LIN {X 0,Y 185.699,Z 175.337,A -85,B 0,C 180,E1 -22153.123,E2 -22153.123} C_VEL
LIN {X 0,Y 185.626,Z 175.353,A -85,B 0,C 180,E1 -22158.819,E2 -22158.819} C_VEL
LIN {X 0,Y 185.544,Z 175.363,A -85,B 0,C 180,E1 -22164.622,E2 -22164.622} C_VEL
LIN {X 0,Y 185.543,Z 175.355,A -85,B 0,C 180,E1 -22169.497,E2 -22169.497} C_VEL
LIN {X 0,Y 185.495,Z 175.376,A -85,B 0,C 180,E1 -22174.631,E2 -22174.631} C_VEL
LIN {X 0,Y 185.497,Z 175.355,A -85,B 0,C 180,E1 -22177.313,E2 -22177.313} C_VEL
LIN {X 0,Y 185.458,Z 175.377,A -85,B 0,C 180,E1 -22180.719,E2 -22180.719} C_VEL
LIN {X 0,Y 185.451,Z 175.371,A -85,B 0,C 180,E1 -22186.055,E2 -22186.055} C_VEL
LIN {X 0,Y 185.452,Z 175.385,A -85,B 0,C 180,E1 -22189.89,E2 -22189.89} C_VEL
LIN {X 0,Y 185.496,Z 175.378,A -85,B 0,C 180,E1 -22192.712,E2 -22192.712} C_VEL
LIN {X 0,Y 185.526,Z 175.377,A -85,B 0,C 180,E1 -22197.971,E2 -22197.971} C_VEL
LIN {X 0,Y 185.542,Z 175.364,A -85,B 0,C 180,E1 -22200.594,E2 -22200.594} C_VEL
LIN {X 0,Y 185.539,Z 175.366,A -85,B 0,C 180,E1 -22205.375,E2 -22205.375} C_VEL
LIN {X 0,Y 185.565,Z 175.425,A -85,B 0,C 180,E1 -22210.242,E2 -22210.242} C_VEL
LIN {X 0,Y 186.59,Z 178.23,A -85,B 0,C 180,E1 -22210.614,E2 -22210.614} C_VEL
LIN {X 0,Y 188.206,Z 180.509,A -85,B 0,C 180,E1 -22211.085,E2 -22211.085} C_VEL
LIN {X 0,Y 196.152,Z 194.206,A -85,B 0,C 180,E1 -22213.376,E2 -22213.376} C_VEL
LIN {X 0,Y 203.397,Z 208.041,A -85,B 0,C 180,E1 -22215.342,E2 -22215.342} C_VEL
LIN {X 0,Y 207.966,Z 220.286,A -85,B 0,C 180,E1 -22216.638,E2 -22216.638} C_VEL
LIN {X 0,Y 204.97,Z 276.924,A -85,B 0,C 180,E1 -22218.566,E2 -22218.566} C_VEL
LIN {X 0,Y 203.672,Z 290.054,A -85,B 0,C 180,E1 -22219.374,E2 -22219.374} C_VEL
LIN {X 0,Y 202.115,Z 302.14,A -85,B 0,C 180,E1 -22220.493,E2 -22220.493} C_VEL
LIN {X 0,Y 200.183,Z 313.622,A -85,B 0,C 180,E1 -22221.927,E2 -22221.927} C_VEL
LIN {X 0,Y 197.643,Z 325.508,A -85,B 0,C 180,E1 -22223.876,E2 -22223.876} C_VEL
LIN {X 0,Y 195.012,Z 336.195,A -85,B 0,C 180,E1 -22226.125,E2 -22226.125} C_VEL
LIN {X 0,Y 192.691,Z 344.89,A -85,B 0,C 180,E1 -22228.432,E2 -22228.432} C_VEL
LIN {X 0,Y 190.067,Z 353.762,A -85,B 0,C 180,E1 -22231.386,E2 -22231.386} C_VEL
LIN {X 0,Y 187.615,Z 361.86,A -85,B 0,C 180,E1 -22234.834,E2 -22234.834} C_VEL
LIN {X 0,Y 186.126,Z 366.937,A -85,B 0,C 180,E1 -22237.594,E2 -22237.594} C_VEL
LIN {X 0,Y 184.688,Z 371.865,A -85,B 0,C 180,E1 -22240.968,E2 -22240.968} C_VEL
LIN {X 0,Y 183.676,Z 375.61,A -85,B 0,C 180,E1 -22244.401,E2 -22244.401} C_VEL
LIN {X 0,Y 183.064,Z 378.261,A -85,B 0,C 180,E1 -22247.886,E2 -22247.886} C_VEL
LIN {X 0,Y 182.859,Z 379.431,A -85,B 0,C 180,E1 -22250.237,E2 -22250.237} C_VEL
LIN {X 0,Y 182.869,Z 380.191,A -85,B 0,C 180,E1 -22252.731,E2 -22252.731} C_VEL
LIN {X 0,Y 182.993,Z 380.465,A -85,B 0,C 180,E1 -22254.99,E2 -22254.99} C_VEL
LIN {X 0,Y 183.532,Z 380.08,A -85,B 0,C 180,E1 -22258.273,E2 -22258.273} C_VEL
LIN {X 0,Y 184.679,Z 378.477,A -85,B 0,C 180,E1 -22262.193,E2 -22262.193} C_VEL
LIN {X 0,Y 186.263,Z 375.796,A -85,B 0,C 180,E1 -22265.791,E2 -22265.791} C_VEL
LIN {X 0,Y 188.446,Z 371.875,A -85,B 0,C 180,E1 -22269.346,E2 -22269.346} C_VEL
LIN {X 0,Y 191.01,Z 366.954,A -85,B 0,C 180,E1 -22272.621,E2 -22272.621} C_VEL
LIN {X 0,Y 194.038,Z 360.951,A -85,B 0,C 180,E1 -22275.671,E2 -22275.671} C_VEL
LIN {X 0,Y 197.307,Z 354.042,A -85,B 0,C 180,E1 -22278.418,E2 -22278.418} C_VEL
LIN {X 0,Y 201.047,Z 345.323,A -85,B 0,C 180,E1 -22281.152,E2 -22281.152} C_VEL
LIN {X 0,Y 204.574,Z 336.068,A -85,B 0,C 180,E1 -22283.42,E2 -22283.42} C_VEL
LIN {X 0,Y 208.06,Z 325.682,A -85,B 0,C 180,E1 -22285.42,E2 -22285.42} C_VEL
LIN {X 0,Y 211.254,Z 314.574,A -85,B 0,C 180,E1 -22287.08,E2 -22287.08} C_VEL
LIN {X 0,Y 213.79,Z 303.24,A -85,B 0,C 180,E1 -22288.392,E2 -22288.392} C_VEL
LIN {X 0,Y 216.105,Z 289.683,A -85,B 0,C 180,E1 -22289.52,E2 -22289.52} C_VEL
LIN {X 0,Y 217.492,Z 277.689,A -85,B 0,C 180,E1 -22290.191,E2 -22290.191} C_VEL
LIN {X 0,Y 220.593,Z 229.858,A -85,B 0,C 180,E1 -22291.736,E2 -22291.736} C_VEL
LIN {X 0,Y 216.192,Z 219.873,A -85,B 0,C 180,E1 -22293.447,E2 -22293.447} C_VEL
LIN {X 0,Y 211.738,Z 211.762,A -85,B 0,C 180,E1 -22295.223,E2 -22295.223} C_VEL
LIN {X 0,Y 206.052,Z 202.859,A -85,B 0,C 180,E1 -22297.65,E2 -22297.65} C_VEL
LIN {X 0,Y 202.931,Z 198.41,A -85,B 0,C 180,E1 -22299.089,E2 -22299.089} C_VEL
LIN {X 0,Y 200.631,Z 195.194,A -85,B 0,C 180,E1 -22300.209,E2 -22300.209} C_VEL
LIN {X 0,Y 197.488,Z 190.877,A -85,B 0,C 180,E1 -22301.859,E2 -22301.859} C_VEL
LIN {X 0,Y 194.917,Z 187.57,A -85,B 0,C 180,E1 -22303.304,E2 -22303.304} C_VEL
LIN {X 0,Y 194.047,Z 186.236,A -85,B 0,C 180,E1 -22303.836,E2 -22303.836} C_VEL
LIN {X 0,Y 191.457,Z 183.668,A -85,B 0,C 180,E1 -22305.384,E2 -22305.384} C_VEL
LIN {X 0,Y 190.076,Z 181.021,A -85,B 0,C 180,E1 -22306.368,E2 -22306.368} C_VEL
LIN {X 0,Y 187.479,Z 179.133,A -85,B 0,C 180,E1 -22308.103,E2 -22308.103} C_VEL
LIN {X 0,Y 186.21,Z 176.799,A -85,B 0,C 180,E1 -22309.174,E2 -22309.174} C_VEL
LIN {X 0,Y 185.915,Z 175.32,A -85,B 0,C 180,E1 -22309.6,E2 -22309.6} C_VEL
LIN {X 0,Y 185.938,Z 175.322,A -85,B 0,C 180,E1 -22313.491,E2 -22313.491} C_VEL
LIN {X 0,Y 186.202,Z 175.284,A -85,B 0,C 180,E1 -22317.839,E2 -22317.839} C_VEL
LIN {X 0,Y 186.395,Z 175.246,A -85,B 0,C 180,E1 -22320.002,E2 -22320.002} C_VEL
LIN {X 0,Y 185.89,Z 175.314,A -85,B 0,C 180,E1 -22324.338,E2 -22324.338} C_VEL
LIN {X 0,Y 185.977,Z 175.315,A -85,B 0,C 180,E1 -22328.696,E2 -22328.696} C_VEL
LIN {X 0,Y 185.716,Z 175.345,A -85,B 0,C 180,E1 -22333.126,E2 -22333.126} C_VEL
LIN {X 0,Y 185.654,Z 175.346,A -85,B 0,C 180,E1 -22337.63,E2 -22337.63} C_VEL
LIN {X 0,Y 185.55,Z 175.357,A -85,B 0,C 180,E1 -22342.259,E2 -22342.259} C_VEL
LIN {X 0,Y 185.503,Z 175.365,A -85,B 0,C 180,E1 -22347.043,E2 -22347.043} C_VEL
LIN {X 0,Y 185.54,Z 175.424,A -85,B 0,C 180,E1 -22349.814,E2 -22349.814} C_VEL
LIN {X 0,Y 186.341,Z 177.863,A -85,B 0,C 180,E1 -22352.539,E2 -22352.539} C_VEL
LIN {X 0,Y 189.581,Z 182.629,A -85,B 0,C 180,E1 -22354.994,E2 -22354.994} C_VEL
LIN {X 0,Y 191.576,Z 185.013,A -85,B 0,C 180,E1 -22356.299,E2 -22356.299} C_VEL
LIN {X 0,Y 195.201,Z 190.145,A -85,B 0,C 180,E1 -22358.541,E2 -22358.541} C_VEL
LIN {X 0,Y 199.91,Z 197.428,A -85,B 0,C 180,E1 -22361.155,E2 -22361.155} C_VEL
LIN {X 0,Y 203.955,Z 204.171,A -85,B 0,C 180,E1 -22363.174,E2 -22363.174} C_VEL
LIN {X 0,Y 210.031,Z 215.033,A -85,B 0,C 180,E1 -22365.927,E2 -22365.927} C_VEL
LIN {X 0,Y 215.137,Z 226.03,A -85,B 0,C 180,E1 -22368.08,E2 -22368.08} C_VEL
LIN {X 0,Y 219.014,Z 236.011,A -85,B 0,C 180,E1 -22369.657,E2 -22369.657} C_VEL
LIN {X 0,Y 219.795,Z 245.363,A -85,B 0,C 180,E1 -22370.312,E2 -22370.312} C_VEL
LIN {X 0,Y 218.586,Z 264.433,A -85,B 0,C 180,E1 -22370.91,E2 -22370.91} C_VEL
LIN {X 0,Y 217.803,Z 270.281,A -85,B 0,C 180,E1 -22370.975,E2 -22370.975} C_VEL
LIN {X 0,Y 212.429,Z 289.298,A -85,B 0,C 180,E1 -22370.579,E2 -22370.579} C_VEL
LIN {X 0,Y 211.21,Z 295.05,A -85,B 0,C 180,E1 -22370.728,E2 -22370.728} C_VEL
LIN {X 0,Y 208.808,Z 308.904,A -85,B 0,C 180,E1 -22371.643,E2 -22371.643} C_VEL
LIN {X 0,Y 206.13,Z 320.49,A -85,B 0,C 180,E1 -22372.758,E2 -22372.758} C_VEL
LIN {X 0,Y 202.791,Z 331.818,A -85,B 0,C 180,E1 -22374.209,E2 -22374.209} C_VEL
LIN {X 0,Y 198.902,Z 343.336,A -85,B 0,C 180,E1 -22376.186,E2 -22376.186} C_VEL
LIN {X 0,Y 194.798,Z 353.604,A -85,B 0,C 180,E1 -22378.457,E2 -22378.457} C_VEL
LIN {X 0,Y 190.425,Z 363.452,A -85,B 0,C 180,E1 -22381.329,E2 -22381.329} C_VEL
LIN {X 0,Y 186.604,Z 371.647,A -85,B 0,C 180,E1 -22384.454,E2 -22384.454} C_VEL
LIN {X 0,Y 183.563,Z 377.81,A -85,B 0,C 180,E1 -22387.489,E2 -22387.489} C_VEL
LIN {X 0,Y 180.871,Z 382.939,A -85,B 0,C 180,E1 -22390.715,E2 -22390.715} C_VEL
LIN {X 0,Y 178.672,Z 386.953,A -85,B 0,C 180,E1 -22394.018,E2 -22394.018} C_VEL
LIN {X 0,Y 176.949,Z 390.71,A -85,B 0,C 180,E1 -22398.546,E2 -22398.546} C_VEL
LIN {X 0,Y 176.403,Z 391.989,A -85,B 0,C 180,E1 -22400.831,E2 -22400.831} C_VEL
LIN {X 0,Y 176.087,Z 392.855,A -85,B 0,C 180,E1 -22403.124,E2 -22403.124} C_VEL
LIN {X 0,Y 175.995,Z 393.414,A -85,B 0,C 180,E1 -22406.709,E2 -22406.709} C_VEL
LIN {X 0,Y 176.204,Z 393.047,A -85,B 0,C 180,E1 -22410,E2 -22410} C_VEL
LIN {X 0,Y 176.009,Z 391.778,A -85,B 0,C 180,E1 -22413.37,E2 -22413.37} C_VEL
LIN {X 0,Y 176.268,Z 388.535,A -85,B 0,C 180,E1 -22418.022,E2 -22418.022} C_VEL
LIN {X 0,Y 176.896,Z 384.919,A -85,B 0,C 180,E1 -22421.458,E2 -22421.458} C_VEL
LIN {X 0,Y 177.989,Z 380.162,A -85,B 0,C 180,E1 -22424.872,E2 -22424.872} C_VEL
LIN {X 0,Y 180.125,Z 373.006,A -85,B 0,C 180,E1 -22428.778,E2 -22428.778} C_VEL
LIN {X 0,Y 182.316,Z 365.664,A -85,B 0,C 180,E1 -22431.887,E2 -22431.887} C_VEL
LIN {X 0,Y 184.764,Z 357.175,A -85,B 0,C 180,E1 -22434.735,E2 -22434.735} C_VEL
LIN {X 0,Y 187.601,Z 347.407,A -85,B 0,C 180,E1 -22437.318,E2 -22437.318} C_VEL
LIN {X 0,Y 190.493,Z 336.558,A -85,B 0,C 180,E1 -22439.568,E2 -22439.568} C_VEL
LIN {X 0,Y 192.977,Z 325.994,A -85,B 0,C 180,E1 -22441.264,E2 -22441.264} C_VEL
LIN {X 0,Y 195.479,Z 313.312,A -85,B 0,C 180,E1 -22442.789,E2 -22442.789} C_VEL
LIN {X 0,Y 197.314,Z 300.667,A -85,B 0,C 180,E1 -22443.894,E2 -22443.894} C_VEL
LIN {X 0,Y 198.573,Z 287.659,A -85,B 0,C 180,E1 -22444.628,E2 -22444.628} C_VEL
LIN {X 0,Y 200.831,Z 240.985,A -85,B 0,C 180,E1 -22446.288,E2 -22446.288} C_VEL
LIN {X 0,Y 198.726,Z 223.599,A -85,B 0,C 180,E1 -22447.42,E2 -22447.42} C_VEL
LIN {X 0,Y 192.377,Z 207.146,A -85,B 0,C 180,E1 -22449.383,E2 -22449.383} C_VEL
LIN {X 0,Y 185.747,Z 192.753,A -85,B 0,C 180,E1 -22451.466,E2 -22451.466} C_VEL
LIN {X 0,Y 180.912,Z 183.531,A -85,B 0,C 180,E1 -22453.042,E2 -22453.042} C_VEL
LIN {X 0,Y 179.45,Z 180.415,A -85,B 0,C 180,E1 -22453.567,E2 -22453.567} C_VEL
LIN {X 0,Y 178.422,Z 176.261,A -85,B 0,C 180,E1 -22456.168,E2 -22456.168} C_VEL
LIN {X 0,Y 178.392,Z 176.267,A -85,B 0,C 180,E1 -22460.923,E2 -22460.923} C_VEL
LIN {X 0,Y 178.489,Z 176.254,A -85,B 0,C 180,E1 -22466.545,E2 -22466.545} C_VEL
LIN {X 0,Y 178.448,Z 176.257,A -85,B 0,C 180,E1 -22471.794,E2 -22471.794} C_VEL
LIN {X 0,Y 178.52,Z 176.248,A -85,B 0,C 180,E1 -22474.888,E2 -22474.888} C_VEL
LIN {X 0,Y 178.61,Z 176.236,A -85,B 0,C 180,E1 -22481.65,E2 -22481.65} C_VEL
LIN {X 0,Y 178.639,Z 176.233,A -85,B 0,C 180,E1 -22486.345,E2 -22486.345} C_VEL
LIN {X 0,Y 178.908,Z 176.173,A -85,B 0,C 180,E1 -22490.958,E2 -22490.958} C_VEL
LIN {X 0,Y 179.128,Z 176.172,A -85,B 0,C 180,E1 -22497.75,E2 -22497.75} C_VEL
LIN {X 0,Y 179.348,Z 176.135,A -85,B 0,C 180,E1 -22499.998,E2 -22499.998} C_VEL
LIN {X 0,Y 178.834,Z 176.177,A -85,B 0,C 180,E1 -22504.506,E2 -22504.506} C_VEL
LIN {X 0,Y 178.907,Z 176.199,A -85,B 0,C 180,E1 -22509.039,E2 -22509.039} C_VEL
LIN {X 0,Y 178.625,Z 176.212,A -85,B 0,C 180,E1 -22513.653,E2 -22513.653} C_VEL
LIN {X 0,Y 178.555,Z 176.234,A -85,B 0,C 180,E1 -22519.15,E2 -22519.15} C_VEL
LIN {X 0,Y 178.464,Z 176.238,A -85,B 0,C 180,E1 -22525.074,E2 -22525.074} C_VEL
LIN {X 0,Y 178.459,Z 176.248,A -85,B 0,C 180,E1 -22530.792,E2 -22530.792} C_VEL
LIN {X 0,Y 178.481,Z 176.25,A -85,B 0,C 180,E1 -22534.216,E2 -22534.216} C_VEL
LIN {X 0,Y 178.384,Z 176.242,A -85,B 0,C 180,E1 -22539.075,E2 -22539.075} C_VEL
LIN {X 0,Y 178.39,Z 176.265,A -85,B 0,C 180,E1 -22542.045,E2 -22542.045} C_VEL
LIN {X 0,Y 178.388,Z 176.257,A -85,B 0,C 180,E1 -22545.163,E2 -22545.163} C_VEL
LIN {X 0,Y 178.393,Z 176.251,A -85,B 0,C 180,E1 -22548.46,E2 -22548.46} C_VEL
LIN {X 0,Y 178.414,Z 176.253,A -85,B 0,C 180,E1 -22553.78,E2 -22553.78} C_VEL
LIN {X 0,Y 178.479,Z 176.248,A -85,B 0,C 180,E1 -22556.544,E2 -22556.544} C_VEL
LIN {X 0,Y 178.434,Z 176.249,A -85,B 0,C 180,E1 -22561.793,E2 -22561.793} C_VEL
LIN {X 0,Y 178.457,Z 176.24,A -85,B 0,C 180,E1 -22566.807,E2 -22566.807} C_VEL
LIN {X 0,Y 178.465,Z 176.276,A -85,B 0,C 180,E1 -22568.576,E2 -22568.576} C_VEL
LIN {X 0,Y 179.41,Z 179.027,A -85,B 0,C 180,E1 -22568.958,E2 -22568.958} C_VEL
LIN {X 0,Y 181.14,Z 181.31,A -85,B 0,C 180,E1 -22569.499,E2 -22569.499} C_VEL
LIN {X 0,Y 189.36,Z 195.188,A -85,B 0,C 180,E1 -22572.042,E2 -22572.042} C_VEL
LIN {X 0,Y 197.797,Z 211.139,A -85,B 0,C 180,E1 -22574.458,E2 -22574.458} C_VEL
LIN {X 0,Y 201.822,Z 222.284,A -85,B 0,C 180,E1 -22575.679,E2 -22575.679} C_VEL
LIN {X 0,Y 198.758,Z 277.285,A -85,B 0,C 180,E1 -22577.595,E2 -22577.595} C_VEL
LIN {X 0,Y 197.404,Z 290.657,A -85,B 0,C 180,E1 -22578.447,E2 -22578.447} C_VEL
LIN {X 0,Y 195.681,Z 303.225,A -85,B 0,C 180,E1 -22579.654,E2 -22579.654} C_VEL
LIN {X 0,Y 193.68,Z 314.47,A -85,B 0,C 180,E1 -22581.128,E2 -22581.128} C_VEL
LIN {X 0,Y 191.164,Z 325.697,A -85,B 0,C 180,E1 -22583.025,E2 -22583.025} C_VEL
LIN {X 0,Y 188.299,Z 336.855,A -85,B 0,C 180,E1 -22585.45,E2 -22585.45} C_VEL
LIN {X 0,Y 185.886,Z 345.472,A -85,B 0,C 180,E1 -22587.833,E2 -22587.833} C_VEL
LIN {X 0,Y 183.36,Z 353.757,A -85,B 0,C 180,E1 -22590.685,E2 -22590.685} C_VEL
LIN {X 0,Y 181.001,Z 361.169,A -85,B 0,C 180,E1 -22593.896,E2 -22593.896} C_VEL
LIN {X 0,Y 179.364,Z 366.428,A -85,B 0,C 180,E1 -22596.75,E2 -22596.75} C_VEL
LIN {X 0,Y 177.796,Z 371.59,A -85,B 0,C 180,E1 -22600.304,E2 -22600.304} C_VEL
LIN {X 0,Y 176.708,Z 375.409,A -85,B 0,C 180,E1 -22603.805,E2 -22603.805} C_VEL
LIN {X 0,Y 176.127,Z 377.76,A -85,B 0,C 180,E1 -22606.738,E2 -22606.738} C_VEL
LIN {X 0,Y 175.766,Z 379.958,A -85,B 0,C 180,E1 -22611.092,E2 -22611.092} C_VEL
LIN {X 0,Y 175.81,Z 380.579,A -85,B 0,C 180,E1 -22613.562,E2 -22613.562} C_VEL
LIN {X 0,Y 176.015,Z 380.698,A -85,B 0,C 180,E1 -22616.053,E2 -22616.053} C_VEL
LIN {X 0,Y 176.555,Z 380.315,A -85,B 0,C 180,E1 -22618.872,E2 -22618.872} C_VEL
LIN {X 0,Y 177.16,Z 379.591,A -85,B 0,C 180,E1 -22621.045,E2 -22621.045} C_VEL
LIN {X 0,Y 178.339,Z 377.895,A -85,B 0,C 180,E1 -22624.154,E2 -22624.154} C_VEL
LIN {X 0,Y 179.921,Z 375.368,A -85,B 0,C 180,E1 -22627.261,E2 -22627.261} C_VEL
LIN {X 0,Y 182.371,Z 371.207,A -85,B 0,C 180,E1 -22630.929,E2 -22630.929} C_VEL
LIN {X 0,Y 185.52,Z 365.487,A -85,B 0,C 180,E1 -22634.59,E2 -22634.59} C_VEL
LIN {X 0,Y 189.483,Z 357.992,A -85,B 0,C 180,E1 -22638.118,E2 -22638.118} C_VEL
LIN {X 0,Y 192.864,Z 350.831,A -85,B 0,C 180,E1 -22640.746,E2 -22640.746} C_VEL
LIN {X 0,Y 196.896,Z 341.505,A -85,B 0,C 180,E1 -22643.428,E2 -22643.428} C_VEL
LIN {X 0,Y 200.615,Z 331.686,A -85,B 0,C 180,E1 -22645.618,E2 -22645.618} C_VEL
LIN {X 0,Y 204.159,Z 320.87,A -85,B 0,C 180,E1 -22647.5,E2 -22647.5} C_VEL
LIN {X 0,Y 207.138,Z 309.895,A -85,B 0,C 180,E1 -22648.983,E2 -22648.983} C_VEL
LIN {X 0,Y 209.576,Z 298.487,A -85,B 0,C 180,E1 -22650.154,E2 -22650.154} C_VEL
LIN {X 0,Y 211.578,Z 285.314,A -85,B 0,C 180,E1 -22651.126,E2 -22651.126} C_VEL
LIN {X 0,Y 212.887,Z 272.862,A -85,B 0,C 180,E1 -22651.687,E2 -22651.687} C_VEL
LIN {X 0,Y 215.494,Z 232.157,A -85,B 0,C 180,E1 -22653.021,E2 -22653.021} C_VEL
LIN {X 0,Y 211.45,Z 223.085,A -85,B 0,C 180,E1 -22654.703,E2 -22654.703} C_VEL
LIN {X 0,Y 207.053,Z 215.086,A -85,B 0,C 180,E1 -22656.578,E2 -22656.578} C_VEL
LIN {X 0,Y 200.756,Z 205.257,A -85,B 0,C 180,E1 -22659.51,E2 -22659.51} C_VEL
LIN {X 0,Y 197.253,Z 200.427,A -85,B 0,C 180,E1 -22661.299,E2 -22661.299} C_VEL
LIN {X 0,Y 194.726,Z 196.808,A -85,B 0,C 180,E1 -22662.713,E2 -22662.713} C_VEL
LIN {X 0,Y 192.016,Z 193.03,A -85,B 0,C 180,E1 -22664.342,E2 -22664.342} C_VEL
LIN {X 0,Y 188.826,Z 189.361,A -85,B 0,C 180,E1 -22666.379,E2 -22666.379} C_VEL
LIN {X 0,Y 187.733,Z 187.466,A -85,B 0,C 180,E1 -22667.194,E2 -22667.194} C_VEL
LIN {X 0,Y 185.167,Z 185.137,A -85,B 0,C 180,E1 -22669.062,E2 -22669.062} C_VEL
LIN {X 0,Y 183.747,Z 182.254,A -85,B 0,C 180,E1 -22670.363,E2 -22670.363} C_VEL
LIN {X 0,Y 180.555,Z 179.962,A -85,B 0,C 180,E1 -22673.156,E2 -22673.156} C_VEL
LIN {X 0,Y 179.168,Z 177.584,A -85,B 0,C 180,E1 -22674.727,E2 -22674.727} C_VEL
LIN {X 0,Y 178.865,Z 176.185,A -85,B 0,C 180,E1 -22675.354,E2 -22675.354} C_VEL
LIN {X 0,Y 179.359,Z 176.122,A -85,B 0,C 180,E1 -22680.002,E2 -22680.002} C_VEL
LIN {X 0,Y 178.899,Z 176.18,A -85,B 0,C 180,E1 -22686.77,E2 -22686.77} C_VEL
LIN {X 0,Y 178.835,Z 176.187,A -85,B 0,C 180,E1 -22690.744,E2 -22690.744} C_VEL
LIN {X 0,Y 178.588,Z 176.221,A -85,B 0,C 180,E1 -22695.992,E2 -22695.992} C_VEL
LIN {X 0,Y 178.555,Z 176.244,A -85,B 0,C 180,E1 -22699.153,E2 -22699.153} C_VEL
LIN {X 0,Y 178.477,Z 176.247,A -85,B 0,C 180,E1 -22705.21,E2 -22705.21} C_VEL
LIN {X 0,Y 178.593,Z 176.951,A -85,B 0,C 180,E1 -22706.122,E2 -22706.122} C_VEL
LIN {X 0,Y 179.564,Z 179.274,A -85,B 0,C 180,E1 -22707.382,E2 -22707.382} C_VEL
LIN {X 0,Y 182.484,Z 182.336,A -85,B 0,C 180,E1 -22710.206,E2 -22710.206} C_VEL
LIN {X 0,Y 184.783,Z 184.988,A -85,B 0,C 180,E1 -22712.175,E2 -22712.175} C_VEL
LIN {X 0,Y 187.569,Z 189.126,A -85,B 0,C 180,E1 -22714.372,E2 -22714.372} C_VEL
LIN {X 0,Y 189.203,Z 191.197,A -85,B 0,C 180,E1 -22715.505,E2 -22715.505} C_VEL
LIN {X 0,Y 193.33,Z 197.395,A -85,B 0,C 180,E1 -22718.171,E2 -22718.171} C_VEL
LIN {X 0,Y 197.052,Z 203.358,A -85,B 0,C 180,E1 -22720.335,E2 -22720.335} C_VEL
LIN {X 0,Y 201.814,Z 211.439,A -85,B 0,C 180,E1 -22722.809,E2 -22722.809} C_VEL
LIN {X 0,Y 207.257,Z 222.099,A -85,B 0,C 180,E1 -22725.408,E2 -22725.408} C_VEL
LIN {X 0,Y 211.553,Z 231.812,A -85,B 0,C 180,E1 -22727.311,E2 -22727.311} C_VEL
LIN {X 0,Y 214.253,Z 239.251,A -85,B 0,C 180,E1 -22728.502,E2 -22728.502} C_VEL
LIN {X 0,Y 214.797,Z 245.776,A -85,B 0,C 180,E1 -22728.991,E2 -22728.991} C_VEL
LIN {X 0,Y 211.832,Z 289.491,A -85,B 0,C 180,E1 -22730.447,E2 -22730.447} C_VEL
LIN {X 0,Y 211.21,Z 295.05,A -85,B 0,C 180,E1 -22730.728,E2 -22730.728} C_VEL
LIN {X 0,Y 209.136,Z 302.593,A -85,B 0,C 180,E1 -22730.948,E2 -22730.948} C_VEL
LIN {X 0,Y 205.966,Z 309.864,A -85,B 0,C 180,E1 -22731.031,E2 -22731.031} C_VEL
LIN {X 0,Y 201.825,Z 318.808,A -85,B 0,C 180,E1 -22731.358,E2 -22731.358} C_VEL
LIN {X 0,Y 199.848,Z 324.061,A -85,B 0,C 180,E1 -22731.829,E2 -22731.829} C_VEL
LIN {X 0,Y 196.647,Z 334.056,A -85,B 0,C 180,E1 -22733.228,E2 -22733.228} C_VEL
LIN {X 0,Y 192.625,Z 345.049,A -85,B 0,C 180,E1 -22735.244,E2 -22735.244} C_VEL
LIN {X 0,Y 188.051,Z 355.788,A -85,B 0,C 180,E1 -22737.821,E2 -22737.821} C_VEL
LIN {X 0,Y 184.229,Z 363.753,A -85,B 0,C 180,E1 -22740.27,E2 -22740.27} C_VEL
LIN {X 0,Y 180.323,Z 371.593,A -85,B 0,C 180,E1 -22743.372,E2 -22743.372} C_VEL
LIN {X 0,Y 177.034,Z 377.893,A -85,B 0,C 180,E1 -22746.611,E2 -22746.611} C_VEL
LIN {X 0,Y 174.173,Z 382.943,A -85,B 0,C 180,E1 -22749.942,E2 -22749.942} C_VEL
LIN {X 0,Y 171.838,Z 386.883,A -85,B 0,C 180,E1 -22753.364,E2 -22753.364} C_VEL
LIN {X 0,Y 169.978,Z 390.573,A -85,B 0,C 180,E1 -22758.07,E2 -22758.07} C_VEL
LIN {X 0,Y 169.37,Z 391.821,A -85,B 0,C 180,E1 -22760.446,E2 -22760.446} C_VEL
LIN {X 0,Y 168.88,Z 393.056,A -85,B 0,C 180,E1 -22765.226,E2 -22765.226} C_VEL
LIN {X 0,Y 168.952,Z 393.095,A -85,B 0,C 180,E1 -22767.616,E2 -22767.616} C_VEL
LIN {X 0,Y 169.106,Z 392.746,A -85,B 0,C 180,E1 -22770,E2 -22770} C_VEL
LIN {X 0,Y 168.934,Z 391.583,A -85,B 0,C 180,E1 -22773.164,E2 -22773.164} C_VEL
LIN {X 0,Y 169.093,Z 389.081,A -85,B 0,C 180,E1 -22777.163,E2 -22777.163} C_VEL
LIN {X 0,Y 169.635,Z 385.757,A -85,B 0,C 180,E1 -22780.745,E2 -22780.745} C_VEL
LIN {X 0,Y 170.604,Z 381.325,A -85,B 0,C 180,E1 -22784.311,E2 -22784.311} C_VEL
LIN {X 0,Y 172.331,Z 375.687,A -85,B 0,C 180,E1 -22787.811,E2 -22787.811} C_VEL
LIN {X 0,Y 174.638,Z 368.618,A -85,B 0,C 180,E1 -22791.235,E2 -22791.235} C_VEL
LIN {X 0,Y 176.736,Z 361.529,A -85,B 0,C 180,E1 -22793.992,E2 -22793.992} C_VEL
LIN {X 0,Y 179.43,Z 352.575,A -85,B 0,C 180,E1 -22796.772,E2 -22796.772} C_VEL
LIN {X 0,Y 182.6,Z 341.774,A -85,B 0,C 180,E1 -22799.389,E2 -22799.389} C_VEL
LIN {X 0,Y 185.409,Z 331.006,A -85,B 0,C 180,E1 -22801.413,E2 -22801.413} C_VEL
LIN {X 0,Y 188.075,Z 318.936,A -85,B 0,C 180,E1 -22803.129,E2 -22803.129} C_VEL
LIN {X 0,Y 190.318,Z 306.404,A -85,B 0,C 180,E1 -22804.435,E2 -22804.435} C_VEL
LIN {X 0,Y 191.956,Z 293.256,A -85,B 0,C 180,E1 -22805.377,E2 -22805.377} C_VEL
LIN {X 0,Y 193.117,Z 275.346,A -85,B 0,C 180,E1 -22806.123,E2 -22806.123} C_VEL
LIN {X 0,Y 194.749,Z 241.728,A -85,B 0,C 180,E1 -22807.338,E2 -22807.338} C_VEL
LIN {X 0,Y 192.871,Z 225.898,A -85,B 0,C 180,E1 -22808.415,E2 -22808.415} C_VEL
LIN {X 0,Y 186.523,Z 209.516,A -85,B 0,C 180,E1 -22810.477,E2 -22810.477} C_VEL
LIN {X 0,Y 180.642,Z 196.638,A -85,B 0,C 180,E1 -22812.437,E2 -22812.437} C_VEL
LIN {X 0,Y 174.152,Z 184.06,A -85,B 0,C 180,E1 -22814.717,E2 -22814.717} C_VEL
LIN {X 0,Y 172.064,Z 180.025,A -85,B 0,C 180,E1 -22815.546,E2 -22815.546} C_VEL
LIN {X 0,Y 171.351,Z 177.143,A -85,B 0,C 180,E1 -22817.586,E2 -22817.586} C_VEL
LIN {X 0,Y 171.365,Z 177.143,A -85,B 0,C 180,E1 -22822.033,E2 -22822.033} C_VEL
LIN {X 0,Y 171.402,Z 177.139,A -85,B 0,C 180,E1 -22825.092,E2 -22825.092} C_VEL
LIN {X 0,Y 171.414,Z 177.134,A -85,B 0,C 180,E1 -22830.526,E2 -22830.526} C_VEL
LIN {X 0,Y 171.441,Z 177.13,A -85,B 0,C 180,E1 -22835.797,E2 -22835.797} C_VEL
LIN {X 0,Y 171.512,Z 177.122,A -85,B 0,C 180,E1 -22840.862,E2 -22840.862} C_VEL
LIN {X 0,Y 171.553,Z 177.114,A -85,B 0,C 180,E1 -22845.769,E2 -22845.769} C_VEL
LIN {X 0,Y 171.847,Z 177.054,A -85,B 0,C 180,E1 -22850.583,E2 -22850.583} C_VEL
LIN {X 0,Y 171.788,Z 177.079,A -85,B 0,C 180,E1 -22855.305,E2 -22855.305} C_VEL
LIN {X 0,Y 172.313,Z 177.011,A -85,B 0,C 180,E1 -22859.998,E2 -22859.998} C_VEL
LIN {X 0,Y 171.845,Z 177.068,A -85,B 0,C 180,E1 -22866.861,E2 -22866.861} C_VEL
LIN {X 0,Y 171.768,Z 177.086,A -85,B 0,C 180,E1 -22870.891,E2 -22870.891} C_VEL
LIN {X 0,Y 171.498,Z 177.089,A -85,B 0,C 180,E1 -22876.668,E2 -22876.668} C_VEL
LIN {X 0,Y 171.479,Z 177.117,A -85,B 0,C 180,E1 -22879.497,E2 -22879.497} C_VEL
LIN {X 0,Y 171.402,Z 177.112,A -85,B 0,C 180,E1 -22885.567,E2 -22885.567} C_VEL
LIN {X 0,Y 171.416,Z 177.124,A -85,B 0,C 180,E1 -22890.57,E2 -22890.57} C_VEL
LIN {X 0,Y 171.39,Z 177.129,A -85,B 0,C 180,E1 -22895.033,E2 -22895.033} C_VEL
LIN {X 0,Y 171.34,Z 177.116,A -85,B 0,C 180,E1 -22898.799,E2 -22898.799} C_VEL
LIN {X 0,Y 171.315,Z 177.145,A -85,B 0,C 180,E1 -22904.216,E2 -22904.216} C_VEL
LIN {X 0,Y 171.326,Z 177.135,A -85,B 0,C 180,E1 -22908.978,E2 -22908.978} C_VEL
LIN {X 0,Y 171.356,Z 177.144,A -85,B 0,C 180,E1 -22912.032,E2 -22912.032} C_VEL
LIN {X 0,Y 171.393,Z 177.122,A -85,B 0,C 180,E1 -22915.091,E2 -22915.091} C_VEL
LIN {X 0,Y 171.403,Z 177.125,A -85,B 0,C 180,E1 -22920.525,E2 -22920.525} C_VEL
LIN {X 0,Y 171.398,Z 177.122,A -85,B 0,C 180,E1 -22925.792,E2 -22925.792} C_VEL
LIN {X 0,Y 171.424,Z 177.115,A -85,B 0,C 180,E1 -22926.749,E2 -22926.749} C_VEL
LIN {X 0,Y 172.488,Z 180.058,A -85,B 0,C 180,E1 -22927.23,E2 -22927.23} C_VEL
LIN {X 0,Y 174.085,Z 182.231,A -85,B 0,C 180,E1 -22927.775,E2 -22927.775} C_VEL
LIN {X 0,Y 181.537,Z 194.391,A -85,B 0,C 180,E1 -22930.264,E2 -22930.264} C_VEL
LIN {X 0,Y 190.267,Z 210.383,A -85,B 0,C 180,E1 -22932.95,E2 -22932.95} C_VEL
LIN {X 0,Y 193.307,Z 217.005,A -85,B 0,C 180,E1 -22933.862,E2 -22933.862} C_VEL
LIN {X 0,Y 195.601,Z 223.464,A -85,B 0,C 180,E1 -22934.598,E2 -22934.598} C_VEL
LIN {X 0,Y 194.287,Z 248.894,A -85,B 0,C 180,E1 -22935.5,E2 -22935.5} C_VEL
LIN {X 0,Y 192.592,Z 277.949,A -85,B 0,C 180,E1 -22936.579,E2 -22936.579} C_VEL
LIN {X 0,Y 191.17,Z 291.281,A -85,B 0,C 180,E1 -22937.459,E2 -22937.459} C_VEL
LIN {X 0,Y 189.291,Z 304.244,A -85,B 0,C 180,E1 -22938.759,E2 -22938.759} C_VEL
LIN {X 0,Y 186.84,Z 316.946,A -85,B 0,C 180,E1 -22940.527,E2 -22940.527} C_VEL
LIN {X 0,Y 184.31,Z 327.672,A -85,B 0,C 180,E1 -22942.472,E2 -22942.472} C_VEL
LIN {X 0,Y 181.629,Z 337.493,A -85,B 0,C 180,E1 -22944.727,E2 -22944.727} C_VEL
LIN {X 0,Y 178.586,Z 347.723,A -85,B 0,C 180,E1 -22947.744,E2 -22947.744} C_VEL
LIN {X 0,Y 175.723,Z 356.532,A -85,B 0,C 180,E1 -22951.062,E2 -22951.062} C_VEL
LIN {X 0,Y 173.333,Z 363.849,A -85,B 0,C 180,E1 -22954.651,E2 -22954.651} C_VEL
LIN {X 0,Y 171.49,Z 369.544,A -85,B 0,C 180,E1 -22958.246,E2 -22958.246} C_VEL
LIN {X 0,Y 170.143,Z 373.984,A -85,B 0,C 180,E1 -22961.919,E2 -22961.919} C_VEL
LIN {X 0,Y 169.482,Z 376.328,A -85,B 0,C 180,E1 -22964.406,E2 -22964.406} C_VEL
LIN {X 0,Y 168.981,Z 378.167,A -85,B 0,C 180,E1 -22966.954,E2 -22966.954} C_VEL
LIN {X 0,Y 168.726,Z 379.532,A -85,B 0,C 180,E1 -22969.464,E2 -22969.464} C_VEL
LIN {X 0,Y 168.736,Z 380.805,A -85,B 0,C 180,E1 -22973.612,E2 -22973.612} C_VEL
LIN {X 0,Y 169.095,Z 380.923,A -85,B 0,C 180,E1 -22977.205,E2 -22977.205} C_VEL
LIN {X 0,Y 169.68,Z 380.464,A -85,B 0,C 180,E1 -22979.803,E2 -22979.803} C_VEL
LIN {X 0,Y 170.478,Z 379.503,A -85,B 0,C 180,E1 -22982.406,E2 -22982.406} C_VEL
LIN {X 0,Y 171.569,Z 378.084,A -85,B 0,C 180,E1 -22984.993,E2 -22984.993} C_VEL
LIN {X 0,Y 173.668,Z 374.961,A -85,B 0,C 180,E1 -22988.831,E2 -22988.831} C_VEL
LIN {X 0,Y 176.449,Z 370.499,A -85,B 0,C 180,E1 -22992.618,E2 -22992.618} C_VEL
LIN {X 0,Y 179.888,Z 364.605,A -85,B 0,C 180,E1 -22996.284,E2 -22996.284} C_VEL
LIN {X 0,Y 184.053,Z 357.058,A -85,B 0,C 180,E1 -22999.791,E2 -22999.791} C_VEL
LIN {X 0,Y 187.81,Z 349.392,A -85,B 0,C 180,E1 -23002.528,E2 -23002.528} C_VEL
LIN {X 0,Y 192.27,Z 339.257,A -85,B 0,C 180,E1 -23005.329,E2 -23005.329} C_VEL
LIN {X 0,Y 196.206,Z 329.061,A -85,B 0,C 180,E1 -23007.503,E2 -23007.503} C_VEL
LIN {X 0,Y 200.033,Z 317.306,A -85,B 0,C 180,E1 -23009.405,E2 -23009.405} C_VEL
LIN {X 0,Y 203.022,Z 305.707,A -85,B 0,C 180,E1 -23010.856,E2 -23010.856} C_VEL
LIN {X 0,Y 205.468,Z 293.49,A -85,B 0,C 180,E1 -23011.975,E2 -23011.975} C_VEL
LIN {X 0,Y 207.19,Z 281.184,A -85,B 0,C 180,E1 -23012.75,E2 -23012.75} C_VEL
LIN {X 0,Y 208.773,Z 261.428,A -85,B 0,C 180,E1 -23013.473,E2 -23013.473} C_VEL
LIN {X 0,Y 210.567,Z 234.613,A -85,B 0,C 180,E1 -23014.357,E2 -23014.357} C_VEL
LIN {X 0,Y 206.546,Z 225.664,A -85,B 0,C 180,E1 -23016.142,E2 -23016.142} C_VEL
LIN {X 0,Y 201.875,Z 217.571,A -85,B 0,C 180,E1 -23018.303,E2 -23018.303} C_VEL
LIN {X 0,Y 197.227,Z 210.262,A -85,B 0,C 180,E1 -23020.636,E2 -23020.636} C_VEL
LIN {X 0,Y 194.111,Z 205.794,A -85,B 0,C 180,E1 -23022.35,E2 -23022.35} C_VEL
LIN {X 0,Y 191.79,Z 202.428,A -85,B 0,C 180,E1 -23023.725,E2 -23023.725} C_VEL
LIN {X 0,Y 188.862,Z 198.425,A -85,B 0,C 180,E1 -23025.592,E2 -23025.592} C_VEL
LIN {X 0,Y 186.253,Z 195.065,A -85,B 0,C 180,E1 -23027.421,E2 -23027.421} C_VEL
LIN {X 0,Y 185.379,Z 193.768,A -85,B 0,C 180,E1 -23028.088,E2 -23028.088} C_VEL
LIN {X 0,Y 182.864,Z 191.052,A -85,B 0,C 180,E1 -23030.086,E2 -23030.086} C_VEL
LIN {X 0,Y 181.508,Z 188.599,A -85,B 0,C 180,E1 -23031.373,E2 -23031.373} C_VEL
LIN {X 0,Y 178.91,Z 186.56,A -85,B 0,C 180,E1 -23033.8,E2 -23033.8} C_VEL
LIN {X 0,Y 177.38,Z 183.784,A -85,B 0,C 180,E1 -23035.692,E2 -23035.692} C_VEL
LIN {X 0,Y 177.125,Z 183.038,A -85,B 0,C 180,E1 -23036.077,E2 -23036.077} C_VEL
LIN {X 0,Y 174.395,Z 181.218,A -85,B 0,C 180,E1 -23039.858,E2 -23039.858} C_VEL
LIN {X 0,Y 172.044,Z 178.214,A -85,B 0,C 180,E1 -23045.569,E2 -23045.569} C_VEL
LIN {X 0,Y 171.846,Z 177.06,A -85,B 0,C 180,E1 -23047.049,E2 -23047.049} C_VEL
LIN {X 0,Y 171.769,Z 177.067,A -85,B 0,C 180,E1 -23050.897,E2 -23050.897} C_VEL
LIN {X 0,Y 171.625,Z 177.195,A -85,B 0,C 180,E1 -23053.621,E2 -23053.621} C_VEL
LIN {X 0,Y 172.47,Z 179.845,A -85,B 0,C 180,E1 -23057.797,E2 -23057.797} C_VEL
LIN {X 0,Y 175.155,Z 182.528,A -85,B 0,C 180,E1 -23062.969,E2 -23062.969} C_VEL
LIN {X 0,Y 176.802,Z 183.241,A -85,B 0,C 180,E1 -23065.115,E2 -23065.115} C_VEL
LIN {X 0,Y 178.176,Z 186.195,A -85,B 0,C 180,E1 -23066.977,E2 -23066.977} C_VEL
LIN {X 0,Y 181.234,Z 189.474,A -85,B 0,C 180,E1 -23070.021,E2 -23070.021} C_VEL
LIN {X 0,Y 182.736,Z 191.304,A -85,B 0,C 180,E1 -23071.362,E2 -23071.362} C_VEL
LIN {X 0,Y 185.532,Z 195.541,A -85,B 0,C 180,E1 -23073.688,E2 -23073.688} C_VEL
LIN {X 0,Y 186.965,Z 197.542,A -85,B 0,C 180,E1 -23074.75,E2 -23074.75} C_VEL
LIN {X 0,Y 190.967,Z 203.794,A -85,B 0,C 180,E1 -23077.474,E2 -23077.474} C_VEL
LIN {X 0,Y 194.259,Z 209.248,A -85,B 0,C 180,E1 -23079.485,E2 -23079.485} C_VEL
LIN {X 0,Y 198.554,Z 216.927,A -85,B 0,C 180,E1 -23081.872,E2 -23081.872} C_VEL
LIN {X 0,Y 203.429,Z 226.706,A -85,B 0,C 180,E1 -23084.342,E2 -23084.342} C_VEL
LIN {X 0,Y 207.289,Z 235.711,A -85,B 0,C 180,E1 -23086.18,E2 -23086.18} C_VEL
LIN {X 0,Y 209.547,Z 241.986,A -85,B 0,C 180,E1 -23087.238,E2 -23087.238} C_VEL
LIN {X 0,Y 209.873,Z 247.469,A -85,B 0,C 180,E1 -23087.631,E2 -23087.631} C_VEL
LIN {X 0,Y 206.937,Z 288.865,A -85,B 0,C 180,E1 -23089.028,E2 -23089.028} C_VEL
LIN {X 0,Y 204.935,Z 302.848,A -85,B 0,C 180,E1 -23089.823,E2 -23089.823} C_VEL
LIN {X 0,Y 202.253,Z 314.964,A -85,B 0,C 180,E1 -23090.803,E2 -23090.803} C_VEL
LIN {X 0,Y 199.848,Z 324.061,A -85,B 0,C 180,E1 -23091.829,E2 -23091.829} C_VEL
LIN {X 0,Y 197.712,Z 329.281,A -85,B 0,C 180,E1 -23092.359,E2 -23092.359} C_VEL
LIN {X 0,Y 192.722,Z 337.523,A -85,B 0,C 180,E1 -23093.081,E2 -23093.081} C_VEL
LIN {X 0,Y 187.525,Z 345.3,A -85,B 0,C 180,E1 -23094.042,E2 -23094.042} C_VEL
LIN {X 0,Y 185.098,Z 349.778,A -85,B 0,C 180,E1 -23094.948,E2 -23094.948} C_VEL
LIN {X 0,Y 180.443,Z 359.529,A -85,B 0,C 180,E1 -23097.62,E2 -23097.62} C_VEL
LIN {X 0,Y 175.967,Z 368.122,A -85,B 0,C 180,E1 -23100.709,E2 -23100.709} C_VEL
LIN {X 0,Y 172.019,Z 375.465,A -85,B 0,C 180,E1 -23104.226,E2 -23104.226} C_VEL
LIN {X 0,Y 168.397,Z 381.425,A -85,B 0,C 180,E1 -23107.938,E2 -23107.938} C_VEL
LIN {X 0,Y 165.806,Z 385.65,A -85,B 0,C 180,E1 -23111.464,E2 -23111.464} C_VEL
LIN {X 0,Y 163.846,Z 388.839,A -85,B 0,C 180,E1 -23115.087,E2 -23115.087} C_VEL
LIN {X 0,Y 162.991,Z 390.45,A -85,B 0,C 180,E1 -23117.55,E2 -23117.55} C_VEL
LIN {X 0,Y 162.358,Z 391.646,A -85,B 0,C 180,E1 -23120.03,E2 -23120.03} C_VEL
LIN {X 0,Y 161.799,Z 392.809,A -85,B 0,C 180,E1 -23125.017,E2 -23125.017} C_VEL
LIN {X 0,Y 161.845,Z 392.82,A -85,B 0,C 180,E1 -23127.512,E2 -23127.512} C_VEL
LIN {X 0,Y 162.012,Z 392.436,A -85,B 0,C 180,E1 -23130.001,E2 -23130.001} C_VEL
LIN {X 0,Y 161.859,Z 391.396,A -85,B 0,C 180,E1 -23132.923,E2 -23132.923} C_VEL
LIN {X 0,Y 162.017,Z 388.664,A -85,B 0,C 180,E1 -23137.478,E2 -23137.478} C_VEL
LIN {X 0,Y 162.615,Z 385.276,A -85,B 0,C 180,E1 -23141.215,E2 -23141.215} C_VEL
LIN {X 0,Y 163.689,Z 380.78,A -85,B 0,C 180,E1 -23144.929,E2 -23144.929} C_VEL
LIN {X 0,Y 165.56,Z 375.071,A -85,B 0,C 180,E1 -23148.565,E2 -23148.565} C_VEL
LIN {X 0,Y 168.005,Z 367.88,A -85,B 0,C 180,E1 -23152.117,E2 -23152.117} C_VEL
LIN {X 0,Y 169.768,Z 362.113,A -85,B 0,C 180,E1 -23154.456,E2 -23154.456} C_VEL
LIN {X 0,Y 172.469,Z 353.582,A -85,B 0,C 180,E1 -23157.286,E2 -23157.286} C_VEL
LIN {X 0,Y 175.684,Z 343.042,A -85,B 0,C 180,E1 -23160.004,E2 -23160.004} C_VEL
LIN {X 0,Y 178.975,Z 331.189,A -85,B 0,C 180,E1 -23162.346,E2 -23162.346} C_VEL
LIN {X 0,Y 181.73,Z 319.262,A -85,B 0,C 180,E1 -23164.109,E2 -23164.109} C_VEL
LIN {X 0,Y 184.066,Z 306.912,A -85,B 0,C 180,E1 -23165.443,E2 -23165.443} C_VEL
LIN {X 0,Y 185.751,Z 294.26,A -85,B 0,C 180,E1 -23166.41,E2 -23166.41} C_VEL
LIN {X 0,Y 186.812,Z 279.809,A -85,B 0,C 180,E1 -23167.076,E2 -23167.076} C_VEL
LIN {X 0,Y 188.739,Z 242.57,A -85,B 0,C 180,E1 -23168.45,E2 -23168.45} C_VEL
LIN {X 0,Y 186.996,Z 228.014,A -85,B 0,C 180,E1 -23169.485,E2 -23169.485} C_VEL
LIN {X 0,Y 180.397,Z 210.983,A -85,B 0,C 180,E1 -23171.76,E2 -23171.76} C_VEL
LIN {X 0,Y 174.04,Z 197.266,A -85,B 0,C 180,E1 -23174.03,E2 -23174.03} C_VEL
LIN {X 0,Y 167.146,Z 184.22,A -85,B 0,C 180,E1 -23176.64,E2 -23176.64} C_VEL
LIN {X 0,Y 164.919,Z 180.186,A -85,B 0,C 180,E1 -23177.529,E2 -23177.529} C_VEL
LIN {X 0,Y 164.67,Z 179.565,A -85,B 0,C 180,E1 -23177.761,E2 -23177.761} C_VEL
LIN {X 0,Y 164.3,Z 178.022,A -85,B 0,C 180,E1 -23178.875,E2 -23178.875} C_VEL
LIN {X 0,Y 164.33,Z 178.018,A -85,B 0,C 180,E1 -23184.35,E2 -23184.35} C_VEL
LIN {X 0,Y 164.375,Z 178.013,A -85,B 0,C 180,E1 -23189.129,E2 -23189.129} C_VEL
LIN {X 0,Y 164.398,Z 178.007,A -85,B 0,C 180,E1 -23194.689,E2 -23194.689} C_VEL
LIN {X 0,Y 164.421,Z 178.002,A -85,B 0,C 180,E1 -23200.116,E2 -23200.116} C_VEL
LIN {X 0,Y 164.482,Z 177.995,A -85,B 0,C 180,E1 -23205.143,E2 -23205.143} C_VEL
LIN {X 0,Y 164.768,Z 177.938,A -85,B 0,C 180,E1 -23210.174,E2 -23210.174} C_VEL
LIN {X 0,Y 164.824,Z 177.922,A -85,B 0,C 180,E1 -23212.649,E2 -23212.649} C_VEL
LIN {X 0,Y 165.277,Z 177.887,A -85,B 0,C 180,E1 -23219.998,E2 -23219.998} C_VEL
LIN {X 0,Y 164.822,Z 177.947,A -85,B 0,C 180,E1 -23227.347,E2 -23227.347} C_VEL
LIN {X 0,Y 164.703,Z 177.966,A -85,B 0,C 180,E1 -23231.056,E2 -23231.056} C_VEL
LIN {X 0,Y 164.423,Z 177.975,A -85,B 0,C 180,E1 -23237.408,E2 -23237.408} C_VEL
LIN {X 0,Y 164.42,Z 177.999,A -85,B 0,C 180,E1 -23239.994,E2 -23239.994} C_VEL
LIN {X 0,Y 164.338,Z 177.986,A -85,B 0,C 180,E1 -23246.092,E2 -23246.092} C_VEL
LIN {X 0,Y 164.356,Z 178.006,A -85,B 0,C 180,E1 -23251.215,E2 -23251.215} C_VEL
LIN {X 0,Y 164.277,Z 177.998,A -85,B 0,C 180,E1 -23256.791,E2 -23256.791} C_VEL
LIN {X 0,Y 164.283,Z 178.003,A -85,B 0,C 180,E1 -23259.916,E2 -23259.916} C_VEL
LIN {X 0,Y 164.277,Z 178.024,A -85,B 0,C 180,E1 -23263.34,E2 -23263.34} C_VEL
LIN {X 0,Y 164.256,Z 178.005,A -85,B 0,C 180,E1 -23266.796,E2 -23266.796} C_VEL
LIN {X 0,Y 164.285,Z 178.023,A -85,B 0,C 180,E1 -23270.353,E2 -23270.353} C_VEL
LIN {X 0,Y 164.321,Z 178.004,A -85,B 0,C 180,E1 -23274.349,E2 -23274.349} C_VEL
LIN {X 0,Y 164.366,Z 178.011,A -85,B 0,C 180,E1 -23279.129,E2 -23279.129} C_VEL
LIN {X 0,Y 164.357,Z 178.008,A -85,B 0,C 180,E1 -23284.766,E2 -23284.766} C_VEL
LIN {X 0,Y 165.285,Z 180.729,A -85,B 0,C 180,E1 -23285.219,E2 -23285.219} C_VEL
LIN {X 0,Y 167.274,Z 183.386,A -85,B 0,C 180,E1 -23285.961,E2 -23285.961} C_VEL
LIN {X 0,Y 176.098,Z 197.581,A -85,B 0,C 180,E1 -23289.116,E2 -23289.116} C_VEL
LIN {X 0,Y 184.31,Z 212.694,A -85,B 0,C 180,E1 -23291.809,E2 -23291.809} C_VEL
LIN {X 0,Y 187.7,Z 219.892,A -85,B 0,C 180,E1 -23292.877,E2 -23292.877} C_VEL
LIN {X 0,Y 189.698,Z 225.655,A -85,B 0,C 180,E1 -23293.554,E2 -23293.554} C_VEL
LIN {X 0,Y 186.516,Z 278.133,A -85,B 0,C 180,E1 -23295.477,E2 -23295.477} C_VEL
LIN {X 0,Y 185.068,Z 291.3,A -85,B 0,C 180,E1 -23296.363,E2 -23296.363} C_VEL
LIN {X 0,Y 183.145,Z 304.173,A -85,B 0,C 180,E1 -23297.675,E2 -23297.675} C_VEL
LIN {X 0,Y 180.769,Z 316.136,A -85,B 0,C 180,E1 -23299.357,E2 -23299.357} C_VEL
LIN {X 0,Y 177.906,Z 327.839,A -85,B 0,C 180,E1 -23301.509,E2 -23301.509} C_VEL
LIN {X 0,Y 174.994,Z 338.094,A -85,B 0,C 180,E1 -23303.948,E2 -23303.948} C_VEL
LIN {X 0,Y 171.832,Z 348.269,A -85,B 0,C 180,E1 -23307.069,E2 -23307.069} C_VEL
LIN {X 0,Y 169.248,Z 355.843,A -85,B 0,C 180,E1 -23310,E2 -23310} C_VEL
LIN {X 0,Y 166.691,Z 363.246,A -85,B 0,C 180,E1 -23313.625,E2 -23313.625} C_VEL
LIN {X 0,Y 164.713,Z 369.105,A -85,B 0,C 180,E1 -23317.354,E2 -23317.354} C_VEL
LIN {X 0,Y 163.256,Z 373.698,A -85,B 0,C 180,E1 -23321.169,E2 -23321.169} C_VEL
LIN {X 0,Y 162.224,Z 377.154,A -85,B 0,C 180,E1 -23325.066,E2 -23325.066} C_VEL
LIN {X 0,Y 161.793,Z 378.871,A -85,B 0,C 180,E1 -23327.702,E2 -23327.702} C_VEL
LIN {X 0,Y 161.6,Z 380.117,A -85,B 0,C 180,E1 -23330.36,E2 -23330.36} C_VEL
LIN {X 0,Y 161.648,Z 381.097,A -85,B 0,C 180,E1 -23334.08,E2 -23334.08} C_VEL
LIN {X 0,Y 162.228,Z 381.105,A -85,B 0,C 180,E1 -23338.459,E2 -23338.459} C_VEL
LIN {X 0,Y 162.93,Z 380.488,A -85,B 0,C 180,E1 -23341.172,E2 -23341.172} C_VEL
LIN {X 0,Y 164.836,Z 378.279,A -85,B 0,C 180,E1 -23345.899,E2 -23345.899} C_VEL
LIN {X 0,Y 166.691,Z 375.703,A -85,B 0,C 180,E1 -23349.229,E2 -23349.229} C_VEL
LIN {X 0,Y 169.578,Z 371.478,A -85,B 0,C 180,E1 -23353.143,E2 -23353.143} C_VEL
LIN {X 0,Y 173.158,Z 365.794,A -85,B 0,C 180,E1 -23356.934,E2 -23356.934} C_VEL
LIN {X 0,Y 176.832,Z 359.614,A -85,B 0,C 180,E1 -23360.059,E2 -23360.059} C_VEL
LIN {X 0,Y 180.641,Z 352.492,A -85,B 0,C 180,E1 -23362.899,E2 -23362.899} C_VEL
LIN {X 0,Y 185.318,Z 342.893,A -85,B 0,C 180,E1 -23365.855,E2 -23365.855} C_VEL
LIN {X 0,Y 189.363,Z 333.393,A -85,B 0,C 180,E1 -23368.1,E2 -23368.1} C_VEL
LIN {X 0,Y 193.514,Z 321.932,A -85,B 0,C 180,E1 -23370.188,E2 -23370.188} C_VEL
LIN {X 0,Y 196.916,Z 310.539,A -85,B 0,C 180,E1 -23371.776,E2 -23371.776} C_VEL
LIN {X 0,Y 199.732,Z 298.296,A -85,B 0,C 180,E1 -23373.05,E2 -23373.05} C_VEL
LIN {X 0,Y 201.843,Z 285.505,A -85,B 0,C 180,E1 -23373.996,E2 -23373.996} C_VEL
LIN {X 0,Y 203.217,Z 273.185,A -85,B 0,C 180,E1 -23374.554,E2 -23374.554} C_VEL
LIN {X 0,Y 205.794,Z 237.248,A -85,B 0,C 180,E1 -23375.736,E2 -23375.736} C_VEL
LIN {X 0,Y 201.978,Z 228.841,A -85,B 0,C 180,E1 -23377.573,E2 -23377.573} C_VEL
LIN {X 0,Y 196.487,Z 219.402,A -85,B 0,C 180,E1 -23380.334,E2 -23380.334} C_VEL
LIN {X 0,Y 191.843,Z 212.23,A -85,B 0,C 180,E1 -23382.96,E2 -23382.96} C_VEL
LIN {X 0,Y 188.524,Z 207.512,A -85,B 0,C 180,E1 -23385.028,E2 -23385.028} C_VEL
LIN {X 0,Y 186.634,Z 204.74,A -85,B 0,C 180,E1 -23386.338,E2 -23386.338} C_VEL
LIN {X 0,Y 183.883,Z 200.995,A -85,B 0,C 180,E1 -23388.379,E2 -23388.379} C_VEL
LIN {X 0,Y 182.789,Z 199.75,A -85,B 0,C 180,E1 -23389.245,E2 -23389.245} C_VEL
LIN {X 0,Y 180.304,Z 196.339,A -85,B 0,C 180,E1 -23391.456,E2 -23391.456} C_VEL
LIN {X 0,Y 179.631,Z 195.2,A -85,B 0,C 180,E1 -23392.131,E2 -23392.131} C_VEL
LIN {X 0,Y 177.116,Z 192.923,A -85,B 0,C 180,E1 -23394.666,E2 -23394.666} C_VEL
LIN {X 0,Y 175.439,Z 189.821,A -85,B 0,C 180,E1 -23396.938,E2 -23396.938} C_VEL
LIN {X 0,Y 171.021,Z 185.192,A -85,B 0,C 180,E1 -23405.899,E2 -23405.899} C_VEL
LIN {X 0,Y 170.85,Z 184.221,A -85,B 0,C 180,E1 -23407.091,E2 -23407.091} C_VEL
LIN {X 0,Y 170.631,Z 184.24,A -85,B 0,C 180,E1 -23413.247,E2 -23413.247} C_VEL
LIN {X 0,Y 173.334,Z 189.076,A -85,B 0,C 180,E1 -23421.649,E2 -23421.649} C_VEL
LIN {X 0,Y 175.393,Z 190.302,A -85,B 0,C 180,E1 -23424.601,E2 -23424.601} C_VEL
LIN {X 0,Y 176.919,Z 193.264,A -85,B 0,C 180,E1 -23426.706,E2 -23426.706} C_VEL
LIN {X 0,Y 179.357,Z 195.878,A -85,B 0,C 180,E1 -23429.234,E2 -23429.234} C_VEL
LIN {X 0,Y 180.735,Z 197.65,A -85,B 0,C 180,E1 -23430.539,E2 -23430.539} C_VEL
LIN {X 0,Y 183.847,Z 202.365,A -85,B 0,C 180,E1 -23433.241,E2 -23433.241} C_VEL
LIN {X 0,Y 188.151,Z 209.352,A -85,B 0,C 180,E1 -23436.43,E2 -23436.43} C_VEL
LIN {X 0,Y 191.424,Z 214.966,A -85,B 0,C 180,E1 -23438.555,E2 -23438.555} C_VEL
LIN {X 0,Y 195.559,Z 222.778,A -85,B 0,C 180,E1 -23441.015,E2 -23441.015} C_VEL
LIN {X 0,Y 199.626,Z 231.188,A -85,B 0,C 180,E1 -23443.202,E2 -23443.202} C_VEL
LIN {X 0,Y 203.233,Z 239.923,A -85,B 0,C 180,E1 -23445.057,E2 -23445.057} C_VEL
LIN {X 0,Y 204.99,Z 245.101,A -85,B 0,C 180,E1 -23445.953,E2 -23445.953} C_VEL
LIN {X 0,Y 205.094,Z 249.221,A -85,B 0,C 180,E1 -23446.219,E2 -23446.219} C_VEL
LIN {X 0,Y 202.094,Z 289.053,A -85,B 0,C 180,E1 -23447.575,E2 -23447.575} C_VEL
LIN {X 0,Y 200.015,Z 302.86,A -85,B 0,C 180,E1 -23448.371,E2 -23448.371} C_VEL
LIN {X 0,Y 197.122,Z 315.374,A -85,B 0,C 180,E1 -23449.408,E2 -23449.408} C_VEL
LIN {X 0,Y 193.481,Z 327.725,A -85,B 0,C 180,E1 -23450.867,E2 -23450.867} C_VEL
LIN {X 0,Y 189.662,Z 338.786,A -85,B 0,C 180,E1 -23452.643,E2 -23452.643} C_VEL
LIN {X 0,Y 185.526,Z 348.817,A -85,B 0,C 180,E1 -23454.712,E2 -23454.712} C_VEL
LIN {X 0,Y 185.098,Z 349.778,A -85,B 0,C 180,E1 -23454.948,E2 -23454.948} C_VEL
LIN {X 0,Y 182.595,Z 354.168,A -85,B 0,C 180,E1 -23455.941,E2 -23455.941} C_VEL
LIN {X 0,Y 176.922,Z 360.926,A -85,B 0,C 180,E1 -23457.408,E2 -23457.408} C_VEL
LIN {X 0,Y 171.18,Z 367.053,A -85,B 0,C 180,E1 -23459.112,E2 -23459.112} C_VEL
LIN {X 0,Y 168.626,Z 370.445,A -85,B 0,C 180,E1 -23460.46,E2 -23460.46} C_VEL
LIN {X 0,Y 164.78,Z 377.075,A -85,B 0,C 180,E1 -23464.008,E2 -23464.008} C_VEL
LIN {X 0,Y 160.867,Z 382.969,A -85,B 0,C 180,E1 -23468.201,E2 -23468.201} C_VEL
LIN {X 0,Y 158.265,Z 386.767,A -85,B 0,C 180,E1 -23471.89,E2 -23471.89} C_VEL
LIN {X 0,Y 156.953,Z 388.749,A -85,B 0,C 180,E1 -23474.416,E2 -23474.416} C_VEL
LIN {X 0,Y 156.021,Z 390.325,A -85,B 0,C 180,E1 -23476.984,E2 -23476.984} C_VEL
LIN {X 0,Y 154.909,Z 392.202,A -85,B 0,C 180,E1 -23482.178,E2 -23482.178} C_VEL
LIN {X 0,Y 154.745,Z 392.544,A -85,B 0,C 180,E1 -23487.397,E2 -23487.397} C_VEL
LIN {X 0,Y 154.919,Z 392.104,A -85,B 0,C 180,E1 -23490.001,E2 -23490.001} C_VEL
LIN {X 0,Y 154.781,Z 391.222,A -85,B 0,C 180,E1 -23492.603,E2 -23492.603} C_VEL
LIN {X 0,Y 154.761,Z 389.933,A -85,B 0,C 180,E1 -23495.212,E2 -23495.212} C_VEL
LIN {X 0,Y 155.149,Z 387.177,A -85,B 0,C 180,E1 -23499.123,E2 -23499.123} C_VEL
LIN {X 0,Y 155.941,Z 383.359,A -85,B 0,C 180,E1 -23503.024,E2 -23503.024} C_VEL
LIN {X 0,Y 157.415,Z 378.395,A -85,B 0,C 180,E1 -23506.871,E2 -23506.871} C_VEL
LIN {X 0,Y 159.516,Z 372.129,A -85,B 0,C 180,E1 -23510.639,E2 -23510.639} C_VEL
LIN {X 0,Y 161.664,Z 365.923,A -85,B 0,C 180,E1 -23513.604,E2 -23513.604} C_VEL
LIN {X 0,Y 164.35,Z 357.979,A -85,B 0,C 180,E1 -23516.681,E2 -23516.681} C_VEL
LIN {X 0,Y 167.431,Z 348.579,A -85,B 0,C 180,E1 -23519.553,E2 -23519.553} C_VEL
LIN {X 0,Y 170.647,Z 338.133,A -85,B 0,C 180,E1 -23522.023,E2 -23522.023} C_VEL
LIN {X 0,Y 173.788,Z 326.549,A -85,B 0,C 180,E1 -23524.133,E2 -23524.133} C_VEL
LIN {X 0,Y 176.565,Z 314.359,A -85,B 0,C 180,E1 -23525.777,E2 -23525.777} C_VEL
LIN {X 0,Y 178.711,Z 301.575,A -85,B 0,C 180,E1 -23527.027,E2 -23527.027} C_VEL
LIN {X 0,Y 180.259,Z 288.304,A -85,B 0,C 180,E1 -23527.885,E2 -23527.885} C_VEL
LIN {X 0,Y 182.749,Z 243.517,A -85,B 0,C 180,E1 -23529.613,E2 -23529.613} C_VEL
LIN {X 0,Y 181.325,Z 230.695,A -85,B 0,C 180,E1 -23530.554,E2 -23530.554} C_VEL
LIN {X 0,Y 175.284,Z 214.753,A -85,B 0,C 180,E1 -23532.781,E2 -23532.781} C_VEL
LIN {X 0,Y 169.304,Z 201.615,A -85,B 0,C 180,E1 -23535.031,E2 -23535.031} C_VEL
LIN {X 0,Y 162.591,Z 188.766,A -85,B 0,C 180,E1 -23537.722,E2 -23537.722} C_VEL
LIN {X 0,Y 159.457,Z 183.397,A -85,B 0,C 180,E1 -23539.044,E2 -23539.044} C_VEL
LIN {X 0,Y 157.697,Z 180.678,A -85,B 0,C 180,E1 -23539.803,E2 -23539.803} C_VEL
LIN {X 0,Y 157.331,Z 179.308,A -85,B 0,C 180,E1 -23540.093,E2 -23540.093} C_VEL
LIN {X 0,Y 157.263,Z 178.899,A -85,B 0,C 180,E1 -23540.473,E2 -23540.473} C_VEL
LIN {X 0,Y 157.279,Z 178.897,A -85,B 0,C 180,E1 -23544.484,E2 -23544.484} C_VEL
LIN {X 0,Y 157.288,Z 178.894,A -85,B 0,C 180,E1 -23548.101,E2 -23548.101} C_VEL
LIN {X 0,Y 157.314,Z 178.891,A -85,B 0,C 180,E1 -23553.462,E2 -23553.462} C_VEL
LIN {X 0,Y 157.364,Z 178.881,A -85,B 0,C 180,E1 -23559.7,E2 -23559.7} C_VEL
LIN {X 0,Y 157.415,Z 178.877,A -85,B 0,C 180,E1 -23564.46,E2 -23564.46} C_VEL
LIN {X 0,Y 157.69,Z 178.823,A -85,B 0,C 180,E1 -23569.729,E2 -23569.729} C_VEL
LIN {X 0,Y 157.762,Z 178.8,A -85,B 0,C 180,E1 -23572.318,E2 -23572.318} C_VEL
LIN {X 0,Y 158.239,Z 178.763,A -85,B 0,C 180,E1 -23579.998,E2 -23579.998} C_VEL
LIN {X 0,Y 157.761,Z 178.828,A -85,B 0,C 180,E1 -23587.678,E2 -23587.678} C_VEL
LIN {X 0,Y 157.632,Z 178.846,A -85,B 0,C 180,E1 -23591.222,E2 -23591.222} C_VEL
LIN {X 0,Y 157.402,Z 178.839,A -85,B 0,C 180,E1 -23595.537,E2 -23595.537} C_VEL
LIN {X 0,Y 157.304,Z 178.889,A -85,B 0,C 180,E1 -23600.94,E2 -23600.94} C_VEL
LIN {X 0,Y 157.265,Z 178.862,A -85,B 0,C 180,E1 -23606.647,E2 -23606.647} C_VEL
LIN {X 0,Y 157.266,Z 178.895,A -85,B 0,C 180,E1 -23612.427,E2 -23612.427} C_VEL
LIN {X 0,Y 157.256,Z 178.874,A -85,B 0,C 180,E1 -23616.442,E2 -23616.442} C_VEL
LIN {X 0,Y 157.187,Z 178.906,A -85,B 0,C 180,E1 -23622.115,E2 -23622.115} C_VEL
LIN {X 0,Y 157.185,Z 178.886,A -85,B 0,C 180,E1 -23627.88,E2 -23627.88} C_VEL
LIN {X 0,Y 157.254,Z 178.888,A -85,B 0,C 180,E1 -23633.554,E2 -23633.554} C_VEL
LIN {X 0,Y 157.278,Z 178.897,A -85,B 0,C 180,E1 -23638.1,E2 -23638.1} C_VEL
LIN {X 0,Y 157.252,Z 178.889,A -85,B 0,C 180,E1 -23642.526,E2 -23642.526} C_VEL
LIN {X 0,Y 158.197,Z 181.653,A -85,B 0,C 180,E1 -23643.031,E2 -23643.031} C_VEL
LIN {X 0,Y 160.283,Z 184.233,A -85,B 0,C 180,E1 -23643.876,E2 -23643.876} C_VEL
LIN {X 0,Y 162.598,Z 187.685,A -85,B 0,C 180,E1 -23644.816,E2 -23644.816} C_VEL
LIN {X 0,Y 171.474,Z 202.219,A -85,B 0,C 180,E1 -23648.191,E2 -23648.191} C_VEL
LIN {X 0,Y 179.183,Z 216.578,A -85,B 0,C 180,E1 -23650.85,E2 -23650.85} C_VEL
LIN {X 0,Y 182.493,Z 223.8,A -85,B 0,C 180,E1 -23651.961,E2 -23651.961} C_VEL
LIN {X 0,Y 183.648,Z 227.074,A -85,B 0,C 180,E1 -23652.374,E2 -23652.374} C_VEL
LIN {X 0,Y 180.473,Z 278.555,A -85,B 0,C 180,E1 -23654.326,E2 -23654.326} C_VEL
LIN {X 0,Y 178.881,Z 292.22,A -85,B 0,C 180,E1 -23655.276,E2 -23655.276} C_VEL
LIN {X 0,Y 176.859,Z 305.024,A -85,B 0,C 180,E1 -23656.645,E2 -23656.645} C_VEL
LIN {X 0,Y 174.382,Z 316.87,A -85,B 0,C 180,E1 -23658.374,E2 -23658.374} C_VEL
LIN {X 0,Y 171.442,Z 328.353,A -85,B 0,C 180,E1 -23660.562,E2 -23660.562} C_VEL
LIN {X 0,Y 168.393,Z 338.643,A -85,B 0,C 180,E1 -23663.108,E2 -23663.108} C_VEL
LIN {X 0,Y 165.092,Z 348.774,A -85,B 0,C 180,E1 -23666.338,E2 -23666.338} C_VEL
LIN {X 0,Y 162.409,Z 356.306,A -85,B 0,C 180,E1 -23669.38,E2 -23669.38} C_VEL
LIN {X 0,Y 159.752,Z 363.658,A -85,B 0,C 180,E1 -23673.152,E2 -23673.152} C_VEL
LIN {X 0,Y 158.002,Z 368.631,A -85,B 0,C 180,E1 -23676.384,E2 -23676.384} C_VEL
LIN {X 0,Y 156.382,Z 373.4,A -85,B 0,C 180,E1 -23680.356,E2 -23680.356} C_VEL
LIN {X 0,Y 155.241,Z 377.009,A -85,B 0,C 180,E1 -23684.417,E2 -23684.417} C_VEL
LIN {X 0,Y 154.594,Z 379.541,A -85,B 0,C 180,E1 -23688.555,E2 -23688.555} C_VEL
LIN {X 0,Y 154.465,Z 380.64,A -85,B 0,C 180,E1 -23691.345,E2 -23691.345} C_VEL
LIN {X 0,Y 154.606,Z 381.381,A -85,B 0,C 180,E1 -23694.618,E2 -23694.618} C_VEL
LIN {X 0,Y 155.437,Z 381.231,A -85,B 0,C 180,E1 -23699.825,E2 -23699.825} C_VEL
LIN {X 0,Y 156.285,Z 380.511,A -85,B 0,C 180,E1 -23702.658,E2 -23702.658} C_VEL
LIN {X 0,Y 158.134,Z 378.474,A -85,B 0,C 180,E1 -23706.876,E2 -23706.876} C_VEL
LIN {X 0,Y 160.652,Z 375.266,A -85,B 0,C 180,E1 -23711.01,E2 -23711.01} C_VEL
LIN {X 0,Y 163.863,Z 370.757,A -85,B 0,C 180,E1 -23715.046,E2 -23715.046} C_VEL
LIN {X 0,Y 167.835,Z 364.813,A -85,B 0,C 180,E1 -23718.915,E2 -23718.915} C_VEL
LIN {X 0,Y 172.008,Z 358.091,A -85,B 0,C 180,E1 -23722.205,E2 -23722.205} C_VEL
LIN {X 0,Y 175.983,Z 350.918,A -85,B 0,C 180,E1 -23724.953,E2 -23724.953} C_VEL
LIN {X 0,Y 180.733,Z 341.327,A -85,B 0,C 180,E1 -23727.789,E2 -23727.789} C_VEL
LIN {X 0,Y 185.311,Z 330.75,A -85,B 0,C 180,E1 -23730.174,E2 -23730.174} C_VEL
LIN {X 0,Y 188.995,Z 320.773,A -85,B 0,C 180,E1 -23731.914,E2 -23731.914} C_VEL
LIN {X 0,Y 192.43,Z 309.255,A -85,B 0,C 180,E1 -23733.482,E2 -23733.482} C_VEL
LIN {X 0,Y 195.44,Z 296.257,A -85,B 0,C 180,E1 -23734.778,E2 -23734.778} C_VEL
LIN {X 0,Y 197.48,Z 283.669,A -85,B 0,C 180,E1 -23735.663,E2 -23735.663} C_VEL
LIN {X 0,Y 198.998,Z 268.764,A -85,B 0,C 180,E1 -23736.246,E2 -23736.246} C_VEL
LIN {X 0,Y 201.175,Z 239.857,A -85,B 0,C 180,E1 -23737.2,E2 -23737.2} C_VEL
LIN {X 0,Y 197.893,Z 232.832,A -85,B 0,C 180,E1 -23738.88,E2 -23738.88} C_VEL
LIN {X 0,Y 192.594,Z 223.522,A -85,B 0,C 180,E1 -23741.777,E2 -23741.777} C_VEL
LIN {X 0,Y 188.6,Z 217.321,A -85,B 0,C 180,E1 -23744.198,E2 -23744.198} C_VEL
LIN {X 0,Y 184.517,Z 211.123,A -85,B 0,C 180,E1 -23747.047,E2 -23747.047} C_VEL
LIN {X 0,Y 181.741,Z 207.212,A -85,B 0,C 180,E1 -23749.224,E2 -23749.224} C_VEL
LIN {X 0,Y 178.585,Z 203.038,A -85,B 0,C 180,E1 -23752.085,E2 -23752.085} C_VEL
LIN {X 0,Y 177.903,Z 201.854,A -85,B 0,C 180,E1 -23752.804,E2 -23752.804} C_VEL
LIN {X 0,Y 175.503,Z 199.418,A -85,B 0,C 180,E1 -23755.408,E2 -23755.408} C_VEL
LIN {X 0,Y 174.043,Z 196.672,A -85,B 0,C 180,E1 -23757.494,E2 -23757.494} C_VEL
LIN {X 0,Y 169.956,Z 191.953,A -85,B 0,C 180,E1 -23766.532,E2 -23766.532} C_VEL
LIN {X 0,Y 169.77,Z 191.163,A -85,B 0,C 180,E1 -23767.903,E2 -23767.903} C_VEL
LIN {X 0,Y 169.657,Z 191.293,A -85,B 0,C 180,E1 -23772.962,E2 -23772.962} C_VEL
LIN {X 0,Y 172.089,Z 195.951,A -85,B 0,C 180,E1 -23781.165,E2 -23781.165} C_VEL
LIN {X 0,Y 173.946,Z 197.103,A -85,B 0,C 180,E1 -23783.973,E2 -23783.973} C_VEL
LIN {X 0,Y 175.685,Z 200.269,A -85,B 0,C 180,E1 -23786.428,E2 -23786.428} C_VEL
LIN {X 0,Y 178.044,Z 202.902,A -85,B 0,C 180,E1 -23788.957,E2 -23788.957} C_VEL
LIN {X 0,Y 179.128,Z 204.621,A -85,B 0,C 180,E1 -23790.056,E2 -23790.056} C_VEL
LIN {X 0,Y 182.342,Z 209.691,A -85,B 0,C 180,E1 -23792.946,E2 -23792.946} C_VEL
LIN {X 0,Y 185.714,Z 215.438,A -85,B 0,C 180,E1 -23795.565,E2 -23795.565} C_VEL
LIN {X 0,Y 188.878,Z 221.156,A -85,B 0,C 180,E1 -23797.757,E2 -23797.757} C_VEL
LIN {X 0,Y 192.697,Z 228.692,A -85,B 0,C 180,E1 -23800.155,E2 -23800.155} C_VEL
LIN {X 0,Y 196.702,Z 237.435,A -85,B 0,C 180,E1 -23802.454,E2 -23802.454} C_VEL
LIN {X 0,Y 200.472,Z 247.509,A -85,B 0,C 180,E1 -23804.521,E2 -23804.521} C_VEL
LIN {X 0,Y 200.542,Z 249.972,A -85,B 0,C 180,E1 -23804.695,E2 -23804.695} C_VEL
LIN {X 0,Y 197.519,Z 288.234,A -85,B 0,C 180,E1 -23805.998,E2 -23805.998} C_VEL
LIN {X 0,Y 195.362,Z 302.285,A -85,B 0,C 180,E1 -23806.808,E2 -23806.808} C_VEL
LIN {X 0,Y 192.402,Z 314.795,A -85,B 0,C 180,E1 -23807.841,E2 -23807.841} C_VEL
LIN {X 0,Y 188.613,Z 327.209,A -85,B 0,C 180,E1 -23809.302,E2 -23809.302} C_VEL
LIN {X 0,Y 185.049,Z 337.047,A -85,B 0,C 180,E1 -23810.847,E2 -23810.847} C_VEL
LIN {X 0,Y 180.74,Z 347.362,A -85,B 0,C 180,E1 -23812.936,E2 -23812.936} C_VEL
LIN {X 0,Y 176.248,Z 356.7,A -85,B 0,C 180,E1 -23815.374,E2 -23815.374} C_VEL
LIN {X 0,Y 171.302,Z 365.753,A -85,B 0,C 180,E1 -23818.46,E2 -23818.46} C_VEL
LIN {X 0,Y 168.626,Z 370.445,A -85,B 0,C 180,E1 -23820.46,E2 -23820.46} C_VEL
LIN {X 0,Y 166.136,Z 373.695,A -85,B 0,C 180,E1 -23821.92,E2 -23821.92} C_VEL
LIN {X 0,Y 160.624,Z 378.483,A -85,B 0,C 180,E1 -23824.274,E2 -23824.274} C_VEL
LIN {X 0,Y 155.26,Z 382.557,A -85,B 0,C 180,E1 -23826.917,E2 -23826.917} C_VEL
LIN {X 0,Y 153.068,Z 384.679,A -85,B 0,C 180,E1 -23828.8,E2 -23828.8} C_VEL
LIN {X 0,Y 150.088,Z 388.67,A -85,B 0,C 180,E1 -23833.683,E2 -23833.683} C_VEL
LIN {X 0,Y 149.077,Z 390.186,A -85,B 0,C 180,E1 -23836.367,E2 -23836.367} C_VEL
LIN {X 0,Y 147.863,Z 391.987,A -85,B 0,C 180,E1 -23841.803,E2 -23841.803} C_VEL
LIN {X 0,Y 147.635,Z 392.318,A -85,B 0,C 180,E1 -23844.537,E2 -23844.537} C_VEL
LIN {X 0,Y 147.693,Z 392.167,A -85,B 0,C 180,E1 -23847.888,E2 -23847.888} C_VEL
LIN {X 0,Y 147.83,Z 391.766,A -85,B 0,C 180,E1 -23850.001,E2 -23850.001} C_VEL
LIN {X 0,Y 147.681,Z 390.852,A -85,B 0,C 180,E1 -23852.728,E2 -23852.728} C_VEL
LIN {X 0,Y 147.692,Z 389.533,A -85,B 0,C 180,E1 -23855.462,E2 -23855.462} C_VEL
LIN {X 0,Y 148.122,Z 386.709,A -85,B 0,C 180,E1 -23859.56,E2 -23859.56} C_VEL
LIN {X 0,Y 148.995,Z 382.82,A -85,B 0,C 180,E1 -23863.642,E2 -23863.642} C_VEL
LIN {X 0,Y 150.595,Z 377.78,A -85,B 0,C 180,E1 -23867.659,E2 -23867.659} C_VEL
LIN {X 0,Y 152.849,Z 371.425,A -85,B 0,C 180,E1 -23871.583,E2 -23871.583} C_VEL
LIN {X 0,Y 154.73,Z 366.285,A -85,B 0,C 180,E1 -23874.13,E2 -23874.13} C_VEL
LIN {X 0,Y 157.98,Z 357.065,A -85,B 0,C 180,E1 -23877.848,E2 -23877.848} C_VEL
LIN {X 0,Y 161.628,Z 346.402,A -85,B 0,C 180,E1 -23881.089,E2 -23881.089} C_VEL
LIN {X 0,Y 165.088,Z 335.57,A -85,B 0,C 180,E1 -23883.603,E2 -23883.603} C_VEL
LIN {X 0,Y 167.947,Z 325.006,A -85,B 0,C 180,E1 -23885.495,E2 -23885.495} C_VEL
LIN {X 0,Y 170.622,Z 313.468,A -85,B 0,C 180,E1 -23887.044,E2 -23887.044} C_VEL
LIN {X 0,Y 172.886,Z 300.115,A -85,B 0,C 180,E1 -23888.355,E2 -23888.355} C_VEL
LIN {X 0,Y 174.372,Z 286.974,A -85,B 0,C 180,E1 -23889.184,E2 -23889.184} C_VEL
LIN {X 0,Y 176.856,Z 244.431,A -85,B 0,C 180,E1 -23890.854,E2 -23890.854} C_VEL
LIN {X 0,Y 175.672,Z 233.051,A -85,B 0,C 180,E1 -23891.721,E2 -23891.721} C_VEL
LIN {X 0,Y 169.785,Z 217.561,A -85,B 0,C 180,E1 -23894.008,E2 -23894.008} C_VEL
LIN {X 0,Y 164.002,Z 204.75,A -85,B 0,C 180,E1 -23896.342,E2 -23896.342} C_VEL
LIN {X 0,Y 158.111,Z 193.293,A -85,B 0,C 180,E1 -23898.863,E2 -23898.863} C_VEL
LIN {X 0,Y 155.007,Z 187.942,A -85,B 0,C 180,E1 -23900.257,E2 -23900.257} C_VEL
LIN {X 0,Y 152.773,Z 184.455,A -85,B 0,C 180,E1 -23901.289,E2 -23901.289} C_VEL
LIN {X 0,Y 150.829,Z 182.014,A -85,B 0,C 180,E1 -23902.187,E2 -23902.187} C_VEL
LIN {X 0,Y 150.171,Z 179.783,A -85,B 0,C 180,E1 -23902.637,E2 -23902.637} C_VEL
LIN {X 0,Y 150.213,Z 179.777,A -85,B 0,C 180,E1 -23907.371,E2 -23907.371} C_VEL
LIN {X 0,Y 150.243,Z 179.77,A -85,B 0,C 180,E1 -23912.721,E2 -23912.721} C_VEL
LIN {X 0,Y 150.288,Z 179.763,A -85,B 0,C 180,E1 -23919.274,E2 -23919.274} C_VEL
LIN {X 0,Y 150.32,Z 179.76,A -85,B 0,C 180,E1 -23923.706,E2 -23923.706} C_VEL
LIN {X 0,Y 150.61,Z 179.709,A -85,B 0,C 180,E1 -23929.24,E2 -23929.24} C_VEL
LIN {X 0,Y 150.685,Z 179.679,A -85,B 0,C 180,E1 -23931.955,E2 -23931.955} C_VEL
LIN {X 0,Y 151.2,Z 179.639,A -85,B 0,C 180,E1 -23939.998,E2 -23939.998} C_VEL
LIN {X 0,Y 150.7,Z 179.709,A -85,B 0,C 180,E1 -23948.04,E2 -23948.04} C_VEL
LIN {X 0,Y 150.575,Z 179.722,A -85,B 0,C 180,E1 -23951.426,E2 -23951.426} C_VEL
LIN {X 0,Y 150.307,Z 179.722,A -85,B 0,C 180,E1 -23956.29,E2 -23956.29} C_VEL
LIN {X 0,Y 150.282,Z 179.764,A -85,B 0,C 180,E1 -23960.72,E2 -23960.72} C_VEL
LIN {X 0,Y 150.183,Z 179.741,A -85,B 0,C 180,E1 -23967.234,E2 -23967.234} C_VEL
LIN {X 0,Y 150.207,Z 179.774,A -85,B 0,C 180,E1 -23972.625,E2 -23972.625} C_VEL
LIN {X 0,Y 150.166,Z 179.749,A -85,B 0,C 180,E1 -23977.472,E2 -23977.472} C_VEL
LIN {X 0,Y 150.13,Z 179.78,A -85,B 0,C 180,E1 -23981.495,E2 -23981.495} C_VEL
LIN {X 0,Y 150.123,Z 179.772,A -85,B 0,C 180,E1 -23985.393,E2 -23985.393} C_VEL
LIN {X 0,Y 150.132,Z 179.772,A -85,B 0,C 180,E1 -23989.051,E2 -23989.051} C_VEL
LIN {X 0,Y 150.171,Z 179.777,A -85,B 0,C 180,E1 -23992.708,E2 -23992.708} C_VEL
LIN {X 0,Y 150.204,Z 179.775,A -85,B 0,C 180,E1 -23997.37,E2 -23997.37} C_VEL
LIN {X 0,Y 150.192,Z 179.786,A -85,B 0,C 180,E1 -24000.029,E2 -24000.029} C_VEL
LIN {X 0,Y 151.053,Z 182.371,A -85,B 0,C 180,E1 -24000.539,E2 -24000.539} C_VEL
LIN {X 0,Y 153.453,Z 185.369,A -85,B 0,C 180,E1 -24001.629,E2 -24001.629} C_VEL
LIN {X 0,Y 155.657,Z 188.672,A -85,B 0,C 180,E1 -24002.628,E2 -24002.628} C_VEL
LIN {X 0,Y 161.293,Z 197.453,A -85,B 0,C 180,E1 -24005.012,E2 -24005.012} C_VEL
LIN {X 0,Y 167.845,Z 208.539,A -85,B 0,C 180,E1 -24007.574,E2 -24007.574} C_VEL
LIN {X 0,Y 175.492,Z 223.292,A -85,B 0,C 180,E1 -24010.328,E2 -24010.328} C_VEL
LIN {X 0,Y 177.489,Z 228.117,A -85,B 0,C 180,E1 -24011.051,E2 -24011.051} C_VEL
LIN {X 0,Y 177.724,Z 230.223,A -85,B 0,C 180,E1 -24011.214,E2 -24011.214} C_VEL
LIN {X 0,Y 174.59,Z 278.213,A -85,B 0,C 180,E1 -24013.054,E2 -24013.054} C_VEL
LIN {X 0,Y 172.939,Z 291.865,A -85,B 0,C 180,E1 -24014.003,E2 -24014.003} C_VEL
LIN {X 0,Y 170.839,Z 304.865,A -85,B 0,C 180,E1 -24015.405,E2 -24015.405} C_VEL
LIN {X 0,Y 168.065,Z 317.596,A -85,B 0,C 180,E1 -24017.317,E2 -24017.317} C_VEL
LIN {X 0,Y 165.006,Z 328.985,A -85,B 0,C 180,E1 -24019.57,E2 -24019.57} C_VEL
LIN {X 0,Y 161.835,Z 339.102,A -85,B 0,C 180,E1 -24022.168,E2 -24022.168} C_VEL
LIN {X 0,Y 158.37,Z 349.282,A -85,B 0,C 180,E1 -24025.545,E2 -24025.545} C_VEL
LIN {X 0,Y 155.581,Z 356.773,A -85,B 0,C 180,E1 -24028.705,E2 -24028.705} C_VEL
LIN {X 0,Y 152.801,Z 364.074,A -85,B 0,C 180,E1 -24032.636,E2 -24032.636} C_VEL
LIN {X 0,Y 150.656,Z 369.876,A -85,B 0,C 180,E1 -24036.697,E2 -24036.697} C_VEL
LIN {X 0,Y 149.08,Z 374.418,A -85,B 0,C 180,E1 -24040.869,E2 -24040.869} C_VEL
LIN {X 0,Y 148.279,Z 376.832,A -85,B 0,C 180,E1 -24043.708,E2 -24043.708} C_VEL
LIN {X 0,Y 147.595,Z 379.374,A -85,B 0,C 180,E1 -24047.77,E2 -24047.77} C_VEL
LIN {X 0,Y 147.378,Z 381.162,A -85,B 0,C 180,E1 -24052.426,E2 -24052.426} C_VEL
LIN {X 0,Y 147.564,Z 381.673,A -85,B 0,C 180,E1 -24055.381,E2 -24055.381} C_VEL
LIN {X 0,Y 147.985,Z 381.735,A -85,B 0,C 180,E1 -24058.353,E2 -24058.353} C_VEL
LIN {X 0,Y 148.864,Z 381.232,A -85,B 0,C 180,E1 -24061.815,E2 -24061.815} C_VEL
LIN {X 0,Y 151.094,Z 379.091,A -85,B 0,C 180,E1 -24067.206,E2 -24067.206} C_VEL
LIN {X 0,Y 153.718,Z 376.073,A -85,B 0,C 180,E1 -24071.524,E2 -24071.524} C_VEL
LIN {X 0,Y 157.083,Z 371.788,A -85,B 0,C 180,E1 -24075.713,E2 -24075.713} C_VEL
LIN {X 0,Y 161.322,Z 365.863,A -85,B 0,C 180,E1 -24079.83,E2 -24079.83} C_VEL
LIN {X 0,Y 166.068,Z 358.669,A -85,B 0,C 180,E1 -24083.521,E2 -24083.521} C_VEL
LIN {X 0,Y 170.605,Z 350.988,A -85,B 0,C 180,E1 -24086.531,E2 -24086.531} C_VEL
LIN {X 0,Y 175.579,Z 341.445,A -85,B 0,C 180,E1 -24089.383,E2 -24089.383} C_VEL
LIN {X 0,Y 180.355,Z 330.929,A -85,B 0,C 180,E1 -24091.776,E2 -24091.776} C_VEL
LIN {X 0,Y 184.378,Z 320.453,A -85,B 0,C 180,E1 -24093.605,E2 -24093.605} C_VEL
LIN {X 0,Y 188.026,Z 308.433,A -85,B 0,C 180,E1 -24095.223,E2 -24095.223} C_VEL
LIN {X 0,Y 191.133,Z 295.383,A -85,B 0,C 180,E1 -24096.487,E2 -24096.487} C_VEL
LIN {X 0,Y 193.182,Z 282.752,A -85,B 0,C 180,E1 -24097.331,E2 -24097.331} C_VEL
LIN {X 0,Y 194.926,Z 264.65,A -85,B 0,C 180,E1 -24098.01,E2 -24098.01} C_VEL
LIN {X 0,Y 196.579,Z 242.39,A -85,B 0,C 180,E1 -24098.786,E2 -24098.786} C_VEL
LIN {X 0,Y 193.067,Z 235.136,A -85,B 0,C 180,E1 -24100.74,E2 -24100.74} C_VEL
LIN {X 0,Y 188.093,Z 226.509,A -85,B 0,C 180,E1 -24103.739,E2 -24103.739} C_VEL
LIN {X 0,Y 183.924,Z 219.896,A -85,B 0,C 180,E1 -24106.624,E2 -24106.624} C_VEL
LIN {X 0,Y 181.609,Z 216.515,A -85,B 0,C 180,E1 -24108.399,E2 -24108.399} C_VEL
LIN {X 0,Y 179.008,Z 212.682,A -85,B 0,C 180,E1 -24110.659,E2 -24110.659} C_VEL
LIN {X 0,Y 176.519,Z 208.997,A -85,B 0,C 180,E1 -24113.142,E2 -24113.142} C_VEL
LIN {X 0,Y 173.392,Z 205.072,A -85,B 0,C 180,E1 -24116.902,E2 -24116.902} C_VEL
LIN {X 0,Y 172.532,Z 203.411,A -85,B 0,C 180,E1 -24118.251,E2 -24118.251} C_VEL
LIN {X 0,Y 168.91,Z 198.732,A -85,B 0,C 180,E1 -24127.173,E2 -24127.173} C_VEL
LIN {X 0,Y 168.837,Z 198.2,A -85,B 0,C 180,E1 -24127.947,E2 -24127.947} C_VEL
LIN {X 0,Y 168.707,Z 198.345,A -85,B 0,C 180,E1 -24132.783,E2 -24132.783} C_VEL
LIN {X 0,Y 170.925,Z 202.865,A -85,B 0,C 180,E1 -24140.793,E2 -24140.793} C_VEL
LIN {X 0,Y 172.533,Z 203.928,A -85,B 0,C 180,E1 -24143.354,E2 -24143.354} C_VEL
LIN {X 0,Y 174.443,Z 207.258,A -85,B 0,C 180,E1 -24146.13,E2 -24146.13} C_VEL
LIN {X 0,Y 176.685,Z 209.871,A -85,B 0,C 180,E1 -24148.623,E2 -24148.623} C_VEL
LIN {X 0,Y 179.6,Z 214.805,A -85,B 0,C 180,E1 -24151.536,E2 -24151.536} C_VEL
LIN {X 0,Y 183.484,Z 221.775,A -85,B 0,C 180,E1 -24154.792,E2 -24154.792} C_VEL
LIN {X 0,Y 186.414,Z 227.392,A -85,B 0,C 180,E1 -24156.964,E2 -24156.964} C_VEL
LIN {X 0,Y 190.682,Z 236.327,A -85,B 0,C 180,E1 -24159.775,E2 -24159.775} C_VEL
LIN {X 0,Y 194.398,Z 245.472,A -85,B 0,C 180,E1 -24162.047,E2 -24162.047} C_VEL
LIN {X 0,Y 196.08,Z 250.178,A -85,B 0,C 180,E1 -24163.027,E2 -24163.027} C_VEL
LIN {X 0,Y 193.225,Z 286.902,A -85,B 0,C 180,E1 -24164.32,E2 -24164.32} C_VEL
LIN {X 0,Y 191.164,Z 300.439,A -85,B 0,C 180,E1 -24165.073,E2 -24165.073} C_VEL
LIN {X 0,Y 188.13,Z 313.324,A -85,B 0,C 180,E1 -24166.097,E2 -24166.097} C_VEL
LIN {X 0,Y 184.474,Z 325.241,A -85,B 0,C 180,E1 -24167.45,E2 -24167.45} C_VEL
LIN {X 0,Y 180.694,Z 335.372,A -85,B 0,C 180,E1 -24168.979,E2 -24168.979} C_VEL
LIN {X 0,Y 175.643,Z 346.966,A -85,B 0,C 180,E1 -24171.303,E2 -24171.303} C_VEL
LIN {X 0,Y 171.347,Z 355.447,A -85,B 0,C 180,E1 -24173.507,E2 -24173.507} C_VEL
LIN {X 0,Y 166.951,Z 363.312,A -85,B 0,C 180,E1 -24176.098,E2 -24176.098} C_VEL
LIN {X 0,Y 162.24,Z 371.052,A -85,B 0,C 180,E1 -24179.404,E2 -24179.404} C_VEL
LIN {X 0,Y 157.702,Z 378.199,A -85,B 0,C 180,E1 -24183.535,E2 -24183.535} C_VEL
LIN {X 0,Y 154.275,Z 383.008,A -85,B 0,C 180,E1 -24187.219,E2 -24187.219} C_VEL
LIN {X 0,Y 153.068,Z 384.679,A -85,B 0,C 180,E1 -24188.8,E2 -24188.8} C_VEL
LIN {X 0,Y 151.014,Z 386.574,A -85,B 0,C 180,E1 -24190.77,E2 -24190.77} C_VEL
LIN {X 0,Y 146.38,Z 389.053,A -85,B 0,C 180,E1 -24194.015,E2 -24194.015} C_VEL
LIN {X 0,Y 142.927,Z 390.482,A -85,B 0,C 180,E1 -24196.791,E2 -24196.791} C_VEL
LIN {X 0,Y 141.299,Z 391.261,A -85,B 0,C 180,E1 -24199.062,E2 -24199.062} C_VEL
LIN {X 0,Y 141.057,Z 391.414,A -85,B 0,C 180,E1 -24199.851,E2 -24199.851} C_VEL
LIN {X 0,Y 140.554,Z 392.074,A -85,B 0,C 180,E1 -24204.261,E2 -24204.261} C_VEL
LIN {X 0,Y 140.618,Z 391.761,A -85,B 0,C 180,E1 -24208.428,E2 -24208.428} C_VEL
LIN {X 0,Y 140.631,Z 390.91,A -85,B 0,C 180,E1 -24211.755,E2 -24211.755} C_VEL
LIN {X 0,Y 140.623,Z 389.129,A -85,B 0,C 180,E1 -24215.737,E2 -24215.737} C_VEL
LIN {X 0,Y 141.086,Z 386.236,A -85,B 0,C 180,E1 -24220.041,E2 -24220.041} C_VEL
LIN {X 0,Y 142.075,Z 382.276,A -85,B 0,C 180,E1 -24224.32,E2 -24224.32} C_VEL
LIN {X 0,Y 144.191,Z 376.162,A -85,B 0,C 180,E1 -24229.209,E2 -24229.209} C_VEL
LIN {X 0,Y 146.766,Z 369.444,A -85,B 0,C 180,E1 -24233.27,E2 -24233.27} C_VEL
LIN {X 0,Y 149.204,Z 362.752,A -85,B 0,C 180,E1 -24236.492,E2 -24236.492} C_VEL
LIN {X 0,Y 152.348,Z 354.293,A -85,B 0,C 180,E1 -24239.731,E2 -24239.731} C_VEL
LIN {X 0,Y 155.9,Z 344.185,A -85,B 0,C 180,E1 -24242.75,E2 -24242.75} C_VEL
LIN {X 0,Y 159.584,Z 332.761,A -85,B 0,C 180,E1 -24245.312,E2 -24245.312} C_VEL
LIN {X 0,Y 162.595,Z 321.548,A -85,B 0,C 180,E1 -24247.239,E2 -24247.239} C_VEL
LIN {X 0,Y 165.425,Z 309.068,A -85,B 0,C 180,E1 -24248.804,E2 -24248.804} C_VEL
LIN {X 0,Y 167.503,Z 296.08,A -85,B 0,C 180,E1 -24249.945,E2 -24249.945} C_VEL
LIN {X 0,Y 168.827,Z 282.333,A -85,B 0,C 180,E1 -24250.713,E2 -24250.713} C_VEL
LIN {X 0,Y 171.045,Z 245.017,A -85,B 0,C 180,E1 -24252.192,E2 -24252.192} C_VEL
LIN {X 0,Y 169.933,Z 235.225,A -85,B 0,C 180,E1 -24252.996,E2 -24252.996} C_VEL
LIN {X 0,Y 164.475,Z 220.558,A -85,B 0,C 180,E1 -24255.274,E2 -24255.274} C_VEL
LIN {X 0,Y 158.891,Z 208.07,A -85,B 0,C 180,E1 -24257.687,E2 -24257.687} C_VEL
LIN {X 0,Y 153.109,Z 196.792,A -85,B 0,C 180,E1 -24260.33,E2 -24260.33} C_VEL
LIN {X 0,Y 150.946,Z 192.984,A -85,B 0,C 180,E1 -24261.375,E2 -24261.375} C_VEL
LIN {X 0,Y 148.477,Z 189.35,A -85,B 0,C 180,E1 -24262.573,E2 -24262.573} C_VEL
LIN {X 0,Y 146.356,Z 185.998,A -85,B 0,C 180,E1 -24263.654,E2 -24263.654} C_VEL
LIN {X 0,Y 143.946,Z 183.253,A -85,B 0,C 180,E1 -24264.867,E2 -24264.867} C_VEL
LIN {X 0,Y 143.132,Z 180.66,A -85,B 0,C 180,E1 -24265.464,E2 -24265.464} C_VEL
LIN {X 0,Y 143.115,Z 180.659,A -85,B 0,C 180,E1 -24270.586,E2 -24270.586} C_VEL
LIN {X 0,Y 143.153,Z 180.654,A -85,B 0,C 180,E1 -24273.776,E2 -24273.776} C_VEL
LIN {X 0,Y 143.251,Z 180.639,A -85,B 0,C 180,E1 -24279.912,E2 -24279.912} C_VEL
LIN {X 0,Y 143.314,Z 180.632,A -85,B 0,C 180,E1 -24285.804,E2 -24285.804} C_VEL
LIN {X 0,Y 143.536,Z 180.595,A -85,B 0,C 180,E1 -24288.703,E2 -24288.703} C_VEL
LIN {X 0,Y 143.61,Z 180.56,A -85,B 0,C 180,E1 -24291.555,E2 -24291.555} C_VEL
LIN {X 0,Y 144.158,Z 180.516,A -85,B 0,C 180,E1 -24299.998,E2 -24299.998} C_VEL
LIN {X 0,Y 143.622,Z 180.593,A -85,B 0,C 180,E1 -24308.439,E2 -24308.439} C_VEL
LIN {X 0,Y 143.499,Z 180.601,A -85,B 0,C 180,E1 -24311.612,E2 -24311.612} C_VEL
LIN {X 0,Y 143.249,Z 180.604,A -85,B 0,C 180,E1 -24317.117,E2 -24317.117} C_VEL
LIN {X 0,Y 143.219,Z 180.644,A -85,B 0,C 180,E1 -24321.191,E2 -24321.191} C_VEL
LIN {X 0,Y 143.14,Z 180.617,A -85,B 0,C 180,E1 -24327.897,E2 -24327.897} C_VEL
LIN {X 0,Y 143.136,Z 180.655,A -85,B 0,C 180,E1 -24333.414,E2 -24333.414} C_VEL
LIN {X 0,Y 143.049,Z 180.641,A -85,B 0,C 180,E1 -24339.691,E2 -24339.691} C_VEL
LIN {X 0,Y 143.048,Z 180.668,A -85,B 0,C 180,E1 -24343.454,E2 -24343.454} C_VEL
LIN {X 0,Y 143.033,Z 180.646,A -85,B 0,C 180,E1 -24347.475,E2 -24347.475} C_VEL
LIN {X 0,Y 143.068,Z 180.668,A -85,B 0,C 180,E1 -24351.807,E2 -24351.807} C_VEL
LIN {X 0,Y 143.164,Z 180.754,A -85,B 0,C 180,E1 -24357.195,E2 -24357.195} C_VEL
LIN {X 0,Y 144.088,Z 183.387,A -85,B 0,C 180,E1 -24357.803,E2 -24357.803} C_VEL
LIN {X 0,Y 146.126,Z 185.571,A -85,B 0,C 180,E1 -24358.823,E2 -24358.823} C_VEL
LIN {X 0,Y 148.562,Z 189.419,A -85,B 0,C 180,E1 -24360.077,E2 -24360.077} C_VEL
LIN {X 0,Y 149.903,Z 191.333,A -85,B 0,C 180,E1 -24360.727,E2 -24360.727} C_VEL
LIN {X 0,Y 155.732,Z 200.181,A -85,B 0,C 180,E1 -24363.407,E2 -24363.407} C_VEL
LIN {X 0,Y 162.724,Z 212.096,A -85,B 0,C 180,E1 -24366.327,E2 -24366.327} C_VEL
LIN {X 0,Y 170.115,Z 226.509,A -85,B 0,C 180,E1 -24369.179,E2 -24369.179} C_VEL
LIN {X 0,Y 171.922,Z 230.855,A -85,B 0,C 180,E1 -24369.868,E2 -24369.868} C_VEL
LIN {X 0,Y 168.637,Z 278.916,A -85,B 0,C 180,E1 -24371.759,E2 -24371.759} C_VEL
LIN {X 0,Y 166.94,Z 292.496,A -85,B 0,C 180,E1 -24372.743,E2 -24372.743} C_VEL
LIN {X 0,Y 164.905,Z 304.596,A -85,B 0,C 180,E1 -24374.076,E2 -24374.076} C_VEL
LIN {X 0,Y 162.216,Z 316.633,A -85,B 0,C 180,E1 -24375.894,E2 -24375.894} C_VEL
LIN {X 0,Y 159.044,Z 328.101,A -85,B 0,C 180,E1 -24378.169,E2 -24378.169} C_VEL
LIN {X 0,Y 155.618,Z 338.705,A -85,B 0,C 180,E1 -24380.905,E2 -24380.905} C_VEL
LIN {X 0,Y 152.3,Z 348.069,A -85,B 0,C 180,E1 -24384.04,E2 -24384.04} C_VEL
LIN {X 0,Y 148.86,Z 356.968,A -85,B 0,C 180,E1 -24387.855,E2 -24387.855} C_VEL
LIN {X 0,Y 145.877,Z 364.463,A -85,B 0,C 180,E1 -24392.07,E2 -24392.07} C_VEL
LIN {X 0,Y 143.31,Z 371.091,A -85,B 0,C 180,E1 -24397.042,E2 -24397.042} C_VEL
LIN {X 0,Y 141.761,Z 375.422,A -85,B 0,C 180,E1 -24401.437,E2 -24401.437} C_VEL
LIN {X 0,Y 140.986,Z 377.666,A -85,B 0,C 180,E1 -24404.432,E2 -24404.432} C_VEL
LIN {X 0,Y 140.47,Z 379.758,A -85,B 0,C 180,E1 -24408.092,E2 -24408.092} C_VEL
LIN {X 0,Y 140.322,Z 381.602,A -85,B 0,C 180,E1 -24413.62,E2 -24413.62} C_VEL
LIN {X 0,Y 140.61,Z 382,A -85,B 0,C 180,E1 -24416.733,E2 -24416.733} C_VEL
LIN {X 0,Y 141.189,Z 381.96,A -85,B 0,C 180,E1 -24419.852,E2 -24419.852} C_VEL
LIN {X 0,Y 142.109,Z 381.403,A -85,B 0,C 180,E1 -24422.956,E2 -24422.956} C_VEL
LIN {X 0,Y 143.336,Z 380.392,A -85,B 0,C 180,E1 -24426.042,E2 -24426.042} C_VEL
LIN {X 0,Y 145.828,Z 377.939,A -85,B 0,C 180,E1 -24430.586,E2 -24430.586} C_VEL
LIN {X 0,Y 149.048,Z 374.277,A -85,B 0,C 180,E1 -24435.014,E2 -24435.014} C_VEL
LIN {X 0,Y 152.981,Z 369.404,A -85,B 0,C 180,E1 -24439.14,E2 -24439.14} C_VEL
LIN {X 0,Y 157.905,Z 362.724,A -85,B 0,C 180,E1 -24443.239,E2 -24443.239} C_VEL
LIN {X 0,Y 162.424,Z 355.901,A -85,B 0,C 180,E1 -24446.401,E2 -24446.401} C_VEL
LIN {X 0,Y 167.188,Z 347.962,A -85,B 0,C 180,E1 -24449.24,E2 -24449.24} C_VEL
LIN {X 0,Y 172.258,Z 338.238,A -85,B 0,C 180,E1 -24451.919,E2 -24451.919} C_VEL
LIN {X 0,Y 176.886,Z 327.901,A -85,B 0,C 180,E1 -24454.086,E2 -24454.086} C_VEL
LIN {X 0,Y 181.002,Z 316.957,A -85,B 0,C 180,E1 -24455.848,E2 -24455.848} C_VEL
LIN {X 0,Y 184.448,Z 305.467,A -85,B 0,C 180,E1 -24457.264,E2 -24457.264} C_VEL
LIN {X 0,Y 187.352,Z 292.374,A -85,B 0,C 180,E1 -24458.439,E2 -24458.439} C_VEL
LIN {X 0,Y 189.386,Z 279.298,A -85,B 0,C 180,E1 -24459.202,E2 -24459.202} C_VEL
LIN {X 0,Y 192.277,Z 245.305,A -85,B 0,C 180,E1 -24460.38,E2 -24460.38} C_VEL
LIN {X 0,Y 188.107,Z 237.075,A -85,B 0,C 180,E1 -24462.917,E2 -24462.917} C_VEL
LIN {X 0,Y 184.187,Z 230.203,A -85,B 0,C 180,E1 -24465.565,E2 -24465.565} C_VEL
LIN {X 0,Y 180.197,Z 223.687,A -85,B 0,C 180,E1 -24468.647,E2 -24468.647} C_VEL
LIN {X 0,Y 177.04,Z 219.029,A -85,B 0,C 180,E1 -24471.505,E2 -24471.505} C_VEL
LIN {X 0,Y 174.335,Z 214.968,A -85,B 0,C 180,E1 -24474.406,E2 -24474.406} C_VEL
LIN {X 0,Y 171.941,Z 211.749,A -85,B 0,C 180,E1 -24477.561,E2 -24477.561} C_VEL
LIN {X 0,Y 171.169,Z 210.218,A -85,B 0,C 180,E1 -24478.844,E2 -24478.844} C_VEL
LIN {X 0,Y 167.917,Z 205.652,A -85,B 0,C 180,E1 -24487.603,E2 -24487.603} C_VEL
LIN {X 0,Y 167.8,Z 205.149,A -85,B 0,C 180,E1 -24488.821,E2 -24488.821} C_VEL
LIN {X 0,Y 167.748,Z 205.385,A -85,B 0,C 180,E1 -24492.475,E2 -24492.475} C_VEL
LIN {X 0,Y 170.038,Z 209.984,A -85,B 0,C 180,E1 -24500.906,E2 -24500.906} C_VEL
LIN {X 0,Y 171.218,Z 210.876,A -85,B 0,C 180,E1 -24502.855,E2 -24502.855} C_VEL
LIN {X 0,Y 173.211,Z 214.261,A -85,B 0,C 180,E1 -24505.835,E2 -24505.835} C_VEL
LIN {X 0,Y 174.968,Z 216.502,A -85,B 0,C 180,E1 -24507.911,E2 -24507.911} C_VEL
LIN {X 0,Y 178.194,Z 222.329,A -85,B 0,C 180,E1 -24511.285,E2 -24511.285} C_VEL
LIN {X 0,Y 181.18,Z 227.932,A -85,B 0,C 180,E1 -24513.915,E2 -24513.915} C_VEL
LIN {X 0,Y 184.496,Z 234.628,A -85,B 0,C 180,E1 -24516.504,E2 -24516.504} C_VEL
LIN {X 0,Y 188.926,Z 244.86,A -85,B 0,C 180,E1 -24519.573,E2 -24519.573} C_VEL
LIN {X 0,Y 191.718,Z 252.655,A -85,B 0,C 180,E1 -24521.401,E2 -24521.401} C_VEL
LIN {X 0,Y 190.586,Z 267.84,A -85,B 0,C 180,E1 -24521.958,E2 -24521.958} C_VEL
LIN {X 0,Y 188.58,Z 289.586,A -85,B 0,C 180,E1 -24522.756,E2 -24522.756} C_VEL
LIN {X 0,Y 186.238,Z 303.044,A -85,B 0,C 180,E1 -24523.56,E2 -24523.56} C_VEL
LIN {X 0,Y 182.819,Z 315.938,A -85,B 0,C 180,E1 -24524.669,E2 -24524.669} C_VEL
LIN {X 0,Y 178.743,Z 327.996,A -85,B 0,C 180,E1 -24526.133,E2 -24526.133} C_VEL
LIN {X 0,Y 174.356,Z 338.826,A -85,B 0,C 180,E1 -24527.924,E2 -24527.924} C_VEL
LIN {X 0,Y 169.697,Z 348.647,A -85,B 0,C 180,E1 -24530.064,E2 -24530.064} C_VEL
LIN {X 0,Y 164.786,Z 357.617,A -85,B 0,C 180,E1 -24532.573,E2 -24532.573} C_VEL
LIN {X 0,Y 159.385,Z 366.411,A -85,B 0,C 180,E1 -24535.792,E2 -24535.792} C_VEL
LIN {X 0,Y 154.718,Z 373.5,A -85,B 0,C 180,E1 -24539.268,E2 -24539.268} C_VEL
LIN {X 0,Y 151.368,Z 378.321,A -85,B 0,C 180,E1 -24542.336,E2 -24542.336} C_VEL
LIN {X 0,Y 147.719,Z 383.049,A -85,B 0,C 180,E1 -24546.147,E2 -24546.147} C_VEL
LIN {X 0,Y 144.795,Z 386.692,A -85,B 0,C 180,E1 -24550.138,E2 -24550.138} C_VEL
LIN {X 0,Y 143.254,Z 388.593,A -85,B 0,C 180,E1 -24552.881,E2 -24552.881} C_VEL
LIN {X 0,Y 141.345,Z 391.1,A -85,B 0,C 180,E1 -24558.529,E2 -24558.529} C_VEL
LIN {X 0,Y 141.057,Z 391.414,A -85,B 0,C 180,E1 -24559.851,E2 -24559.851} C_VEL
LIN {X 0,Y 140.059,Z 391.899,A -85,B 0,C 180,E1 -24562.219,E2 -24562.219} C_VEL
LIN {X 0,Y 138.329,Z 391.994,A -85,B 0,C 180,E1 -24564.56,E2 -24564.56} C_VEL
LIN {X 0,Y 134.604,Z 391.294,A -85,B 0,C 180,E1 -24569.345,E2 -24569.345} C_VEL
LIN {X 0,Y 133.494,Z 390.215,A -85,B 0,C 180,E1 -24572.7,E2 -24572.7} C_VEL
LIN {X 0,Y 133.55,Z 388.7,A -85,B 0,C 180,E1 -24576.042,E2 -24576.042} C_VEL
LIN {X 0,Y 134.076,Z 385.741,A -85,B 0,C 180,E1 -24580.572,E2 -24580.572} C_VEL
LIN {X 0,Y 135.165,Z 381.701,A -85,B 0,C 180,E1 -24585.07,E2 -24585.07} C_VEL
LIN {X 0,Y 137.457,Z 375.463,A -85,B 0,C 180,E1 -24590.19,E2 -24590.19} C_VEL
LIN {X 0,Y 140.253,Z 368.652,A -85,B 0,C 180,E1 -24594.42,E2 -24594.42} C_VEL
LIN {X 0,Y 142.482,Z 362.707,A -85,B 0,C 180,E1 -24597.39,E2 -24597.39} C_VEL
LIN {X 0,Y 146.192,Z 353.259,A -85,B 0,C 180,E1 -24601.118,E2 -24601.118} C_VEL
LIN {X 0,Y 149.977,Z 342.923,A -85,B 0,C 180,E1 -24604.218,E2 -24604.218} C_VEL
LIN {X 0,Y 153.805,Z 331.263,A -85,B 0,C 180,E1 -24606.852,E2 -24606.852} C_VEL
LIN {X 0,Y 156.994,Z 319.745,A -85,B 0,C 180,E1 -24608.81,E2 -24608.81} C_VEL
LIN {X 0,Y 159.7,Z 307.875,A -85,B 0,C 180,E1 -24610.269,E2 -24610.269} C_VEL
LIN {X 0,Y 161.801,Z 294.793,A -85,B 0,C 180,E1 -24611.417,E2 -24611.417} C_VEL
LIN {X 0,Y 163.023,Z 282.422,A -85,B 0,C 180,E1 -24612.11,E2 -24612.11} C_VEL
LIN {X 0,Y 165.305,Z 245.802,A -85,B 0,C 180,E1 -24613.594,E2 -24613.594} C_VEL
LIN {X 0,Y 164.335,Z 237.509,A -85,B 0,C 180,E1 -24614.328,E2 -24614.328} C_VEL
LIN {X 0,Y 159.099,Z 223.197,A -85,B 0,C 180,E1 -24616.691,E2 -24616.691} C_VEL
LIN {X 0,Y 153.092,Z 209.812,A -85,B 0,C 180,E1 -24619.466,E2 -24619.466} C_VEL
LIN {X 0,Y 147.343,Z 198.545,A -85,B 0,C 180,E1 -24622.358,E2 -24622.358} C_VEL
LIN {X 0,Y 144.287,Z 194.133,A -85,B 0,C 180,E1 -24623.903,E2 -24623.903} C_VEL
LIN {X 0,Y 141.93,Z 190.658,A -85,B 0,C 180,E1 -24625.177,E2 -24625.177} C_VEL
LIN {X 0,Y 139.86,Z 187.751,A -85,B 0,C 180,E1 -24626.348,E2 -24626.348} C_VEL
LIN {X 0,Y 139.126,Z 186.495,A -85,B 0,C 180,E1 -24626.796,E2 -24626.796} C_VEL
LIN {X 0,Y 136.968,Z 184.19,A -85,B 0,C 180,E1 -24628.049,E2 -24628.049} C_VEL
LIN {X 0,Y 136.056,Z 181.54,A -85,B 0,C 180,E1 -24628.788,E2 -24628.788} C_VEL
LIN {X 0,Y 136.144,Z 181.527,A -85,B 0,C 180,E1 -24632.313,E2 -24632.313} C_VEL
LIN {X 0,Y 136.194,Z 181.52,A -85,B 0,C 180,E1 -24638.822,E2 -24638.822} C_VEL
LIN {X 0,Y 136.231,Z 181.514,A -85,B 0,C 180,E1 -24645.049,E2 -24645.049} C_VEL
LIN {X 0,Y 136.429,Z 181.484,A -85,B 0,C 180,E1 -24648.176,E2 -24648.176} C_VEL
LIN {X 0,Y 136.54,Z 181.441,A -85,B 0,C 180,E1 -24651.115,E2 -24651.115} C_VEL
LIN {X 0,Y 137.115,Z 181.392,A -85,B 0,C 180,E1 -24659.998,E2 -24659.998} C_VEL
LIN {X 0,Y 136.548,Z 181.476,A -85,B 0,C 180,E1 -24668.88,E2 -24668.88} C_VEL
LIN {X 0,Y 136.414,Z 181.481,A -85,B 0,C 180,E1 -24671.89,E2 -24671.89} C_VEL
LIN {X 0,Y 136.162,Z 181.494,A -85,B 0,C 180,E1 -24678.038,E2 -24678.038} C_VEL
LIN {X 0,Y 136.143,Z 181.527,A -85,B 0,C 180,E1 -24681.687,E2 -24681.687} C_VEL
LIN {X 0,Y 136.06,Z 181.5,A -85,B 0,C 180,E1 -24688.583,E2 -24688.583} C_VEL
LIN {X 0,Y 136.038,Z 181.532,A -85,B 0,C 180,E1 -24694.627,E2 -24694.627} C_VEL
LIN {X 0,Y 136.021,Z 181.512,A -85,B 0,C 180,E1 -24699.191,E2 -24699.191} C_VEL
LIN {X 0,Y 135.99,Z 181.546,A -85,B 0,C 180,E1 -24703.653,E2 -24703.653} C_VEL
LIN {X 0,Y 135.978,Z 181.524,A -85,B 0,C 180,E1 -24707.785,E2 -24707.785} C_VEL
LIN {X 0,Y 136.043,Z 181.526,A -85,B 0,C 180,E1 -24713.792,E2 -24713.792} C_VEL
LIN {X 0,Y 136.957,Z 184.272,A -85,B 0,C 180,E1 -24714.555,E2 -24714.555} C_VEL
LIN {X 0,Y 139.008,Z 186.458,A -85,B 0,C 180,E1 -24715.74,E2 -24715.74} C_VEL
LIN {X 0,Y 139.562,Z 186.998,A -85,B 0,C 180,E1 -24716.049,E2 -24716.049} C_VEL
LIN {X 0,Y 141.527,Z 190.211,A -85,B 0,C 180,E1 -24717.211,E2 -24717.211} C_VEL
LIN {X 0,Y 143.073,Z 192.182,A -85,B 0,C 180,E1 -24718.043,E2 -24718.043} C_VEL
LIN {X 0,Y 148.798,Z 200.711,A -85,B 0,C 180,E1 -24720.966,E2 -24720.966} C_VEL
LIN {X 0,Y 155.6,Z 211.942,A -85,B 0,C 180,E1 -24724.122,E2 -24724.122} C_VEL
LIN {X 0,Y 162.13,Z 224.226,A -85,B 0,C 180,E1 -24726.878,E2 -24726.878} C_VEL
LIN {X 0,Y 166.147,Z 232.595,A -85,B 0,C 180,E1 -24728.483,E2 -24728.483} C_VEL
LIN {X 0,Y 162.912,Z 278.496,A -85,B 0,C 180,E1 -24730.321,E2 -24730.321} C_VEL
LIN {X 0,Y 161.115,Z 292.338,A -85,B 0,C 180,E1 -24731.323,E2 -24731.323} C_VEL
LIN {X 0,Y 158.844,Z 305.298,A -85,B 0,C 180,E1 -24732.789,E2 -24732.789} C_VEL
LIN {X 0,Y 156.02,Z 317.246,A -85,B 0,C 180,E1 -24734.654,E2 -24734.654} C_VEL
LIN {X 0,Y 152.745,Z 328.548,A -85,B 0,C 180,E1 -24736.973,E2 -24736.973} C_VEL
LIN {X 0,Y 149.155,Z 339.179,A -85,B 0,C 180,E1 -24739.822,E2 -24739.822} C_VEL
LIN {X 0,Y 145.674,Z 348.511,A -85,B 0,C 180,E1 -24743.072,E2 -24743.072} C_VEL
LIN {X 0,Y 141.984,Z 357.617,A -85,B 0,C 180,E1 -24747.162,E2 -24747.162} C_VEL
LIN {X 0,Y 138.974,Z 364.835,A -85,B 0,C 180,E1 -24751.448,E2 -24751.448} C_VEL
LIN {X 0,Y 136.602,Z 370.596,A -85,B 0,C 180,E1 -24755.905,E2 -24755.905} C_VEL
LIN {X 0,Y 134.94,Z 374.963,A -85,B 0,C 180,E1 -24760.351,E2 -24760.351} C_VEL
LIN {X 0,Y 133.735,Z 378.463,A -85,B 0,C 180,E1 -24765.233,E2 -24765.233} C_VEL
LIN {X 0,Y 133.34,Z 380.13,A -85,B 0,C 180,E1 -24768.435,E2 -24768.435} C_VEL
LIN {X 0,Y 133.152,Z 381.295,A -85,B 0,C 180,E1 -24771.682,E2 -24771.682} C_VEL
LIN {X 0,Y 133.477,Z 382.209,A -85,B 0,C 180,E1 -24776.484,E2 -24776.484} C_VEL
LIN {X 0,Y 134.507,Z 382.1,A -85,B 0,C 180,E1 -24781.5,E2 -24781.5} C_VEL
LIN {X 0,Y 135.614,Z 381.438,A -85,B 0,C 180,E1 -24784.754,E2 -24784.754} C_VEL
LIN {X 0,Y 138.442,Z 379.072,A -85,B 0,C 180,E1 -24790.41,E2 -24790.41} C_VEL
LIN {X 0,Y 141.031,Z 376.478,A -85,B 0,C 180,E1 -24794.239,E2 -24794.239} C_VEL
LIN {X 0,Y 144.983,Z 372.141,A -85,B 0,C 180,E1 -24798.708,E2 -24798.708} C_VEL
LIN {X 0,Y 149.695,Z 366.359,A -85,B 0,C 180,E1 -24802.952,E2 -24802.952} C_VEL
LIN {X 0,Y 154.468,Z 360.007,A -85,B 0,C 180,E1 -24806.399,E2 -24806.399} C_VEL
LIN {X 0,Y 159.223,Z 352.876,A -85,B 0,C 180,E1 -24809.397,E2 -24809.397} C_VEL
LIN {X 0,Y 164.456,Z 344.097,A -85,B 0,C 180,E1 -24812.235,E2 -24812.235} C_VEL
LIN {X 0,Y 169.283,Z 334.786,A -85,B 0,C 180,E1 -24814.552,E2 -24814.552} C_VEL
LIN {X 0,Y 174.098,Z 323.867,A -85,B 0,C 180,E1 -24816.612,E2 -24816.612} C_VEL
LIN {X 0,Y 177.911,Z 313.255,A -85,B 0,C 180,E1 -24818.174,E2 -24818.174} C_VEL
LIN {X 0,Y 181.424,Z 301.038,A -85,B 0,C 180,E1 -24819.517,E2 -24819.517} C_VEL
LIN {X 0,Y 184.057,Z 288.223,A -85,B 0,C 180,E1 -24820.517,E2 -24820.517} C_VEL
LIN {X 0,Y 185.825,Z 275.318,A -85,B 0,C 180,E1 -24821.137,E2 -24821.137} C_VEL
LIN {X 0,Y 188.109,Z 248.424,A -85,B 0,C 180,E1 -24822.062,E2 -24822.062} C_VEL
LIN {X 0,Y 183.414,Z 239.153,A -85,B 0,C 180,E1 -24825.242,E2 -24825.242} C_VEL
LIN {X 0,Y 179.004,Z 231.553,A -85,B 0,C 180,E1 -24828.681,E2 -24828.681} C_VEL
LIN {X 0,Y 175.307,Z 225.601,A -85,B 0,C 180,E1 -24832.173,E2 -24832.173} C_VEL
LIN {X 0,Y 172.712,Z 221.566,A -85,B 0,C 180,E1 -24835.141,E2 -24835.141} C_VEL
LIN {X 0,Y 170.308,Z 217.981,A -85,B 0,C 180,E1 -24838.584,E2 -24838.584} C_VEL
LIN {X 0,Y 169.876,Z 217.02,A -85,B 0,C 180,E1 -24839.372,E2 -24839.372} C_VEL
LIN {X 0,Y 166.933,Z 212.572,A -85,B 0,C 180,E1 -24848.039,E2 -24848.039} C_VEL
LIN {X 0,Y 166.873,Z 212.159,A -85,B 0,C 180,E1 -24848.87,E2 -24848.87} C_VEL
LIN {X 0,Y 166.796,Z 212.404,A -85,B 0,C 180,E1 -24852.164,E2 -24852.164} C_VEL
LIN {X 0,Y 168.897,Z 216.912,A -85,B 0,C 180,E1 -24860.526,E2 -24860.526} C_VEL
LIN {X 0,Y 169.914,Z 217.777,A -85,B 0,C 180,E1 -24862.334,E2 -24862.334} C_VEL
LIN {X 0,Y 171.97,Z 221.206,A -85,B 0,C 180,E1 -24865.512,E2 -24865.512} C_VEL
LIN {X 0,Y 173.35,Z 223.283,A -85,B 0,C 180,E1 -24867.273,E2 -24867.273} C_VEL
LIN {X 0,Y 176.137,Z 228.514,A -85,B 0,C 180,E1 -24870.365,E2 -24870.365} C_VEL
LIN {X 0,Y 179.097,Z 234.41,A -85,B 0,C 180,E1 -24873.169,E2 -24873.169} C_VEL
LIN {X 0,Y 182.788,Z 242.519,A -85,B 0,C 180,E1 -24876.202,E2 -24876.202} C_VEL
LIN {X 0,Y 186.443,Z 251.839,A -85,B 0,C 180,E1 -24878.894,E2 -24878.894} C_VEL
LIN {X 0,Y 187.622,Z 255.359,A -85,B 0,C 180,E1 -24879.729,E2 -24879.729} C_VEL
LIN {X 0,Y 184.712,Z 287.951,A -85,B 0,C 180,E1 -24880.892,E2 -24880.892} C_VEL
LIN {X 0,Y 182.352,Z 301.621,A -85,B 0,C 180,E1 -24881.686,E2 -24881.686} C_VEL
LIN {X 0,Y 179.197,Z 313.674,A -85,B 0,C 180,E1 -24882.662,E2 -24882.662} C_VEL
LIN {X 0,Y 174.952,Z 326.111,A -85,B 0,C 180,E1 -24884.106,E2 -24884.106} C_VEL
LIN {X 0,Y 170.838,Z 335.976,A -85,B 0,C 180,E1 -24885.625,E2 -24885.625} C_VEL
LIN {X 0,Y 165.432,Z 347.336,A -85,B 0,C 180,E1 -24888.003,E2 -24888.003} C_VEL
LIN {X 0,Y 160.223,Z 356.487,A -85,B 0,C 180,E1 -24890.504,E2 -24890.504} C_VEL
LIN {X 0,Y 154.478,Z 365.425,A -85,B 0,C 180,E1 -24893.741,E2 -24893.741} C_VEL
LIN {X 0,Y 149.409,Z 372.656,A -85,B 0,C 180,E1 -24897.252,E2 -24897.252} C_VEL
LIN {X 0,Y 145.113,Z 378.48,A -85,B 0,C 180,E1 -24901.033,E2 -24901.033} C_VEL
LIN {X 0,Y 141.226,Z 383.109,A -85,B 0,C 180,E1 -24904.977,E2 -24904.977} C_VEL
LIN {X 0,Y 138.113,Z 386.664,A -85,B 0,C 180,E1 -24909.134,E2 -24909.134} C_VEL
LIN {X 0,Y 136.45,Z 388.495,A -85,B 0,C 180,E1 -24911.999,E2 -24911.999} C_VEL
LIN {X 0,Y 134.356,Z 390.924,A -85,B 0,C 180,E1 -24917.923,E2 -24917.923} C_VEL
LIN {X 0,Y 133.795,Z 391.567,A -85,B 0,C 180,E1 -24920.934,E2 -24920.934} C_VEL
LIN {X 0,Y 133.469,Z 391.814,A -85,B 0,C 180,E1 -24923.955,E2 -24923.955} C_VEL
LIN {X 0,Y 133.557,Z 391.328,A -85,B 0,C 180,E1 -24929.006,E2 -24929.006} C_VEL
LIN {X 0,Y 133.494,Z 390.215,A -85,B 0,C 180,E1 -24932.7,E2 -24932.7} C_VEL
LIN {X 0,Y 133.183,Z 389.524,A -85,B 0,C 180,E1 -24934.359,E2 -24934.359} C_VEL
LIN {X 0,Y 131.422,Z 387.723,A -85,B 0,C 180,E1 -24937.606,E2 -24937.606} C_VEL
LIN {X 0,Y 128.456,Z 384.175,A -85,B 0,C 180,E1 -24942.479,E2 -24942.479} C_VEL
LIN {X 0,Y 128.051,Z 382.001,A -85,B 0,C 180,E1 -24944.958,E2 -24944.958} C_VEL
LIN {X 0,Y 128.223,Z 381.214,A -85,B 0,C 180,E1 -24945.777,E2 -24945.777} C_VEL
LIN {X 0,Y 130.784,Z 374.766,A -85,B 0,C 180,E1 -24951.269,E2 -24951.269} C_VEL
LIN {X 0,Y 133.775,Z 367.865,A -85,B 0,C 180,E1 -24955.68,E2 -24955.68} C_VEL
LIN {X 0,Y 135.845,Z 362.579,A -85,B 0,C 180,E1 -24958.413,E2 -24958.413} C_VEL
LIN {X 0,Y 139.371,Z 354.023,A -85,B 0,C 180,E1 -24961.971,E2 -24961.971} C_VEL
LIN {X 0,Y 143.253,Z 343.973,A -85,B 0,C 180,E1 -24965.202,E2 -24965.202} C_VEL
LIN {X 0,Y 147.239,Z 332.632,A -85,B 0,C 180,E1 -24967.92,E2 -24967.92} C_VEL
LIN {X 0,Y 150.496,Z 321.508,A -85,B 0,C 180,E1 -24969.95,E2 -24969.95} C_VEL
LIN {X 0,Y 153.536,Z 309.222,A -85,B 0,C 180,E1 -24971.586,E2 -24971.586} C_VEL
LIN {X 0,Y 155.829,Z 296.154,A -85,B 0,C 180,E1 -24972.802,E2 -24972.802} C_VEL
LIN {X 0,Y 157.315,Z 282.539,A -85,B 0,C 180,E1 -24973.606,E2 -24973.606} C_VEL
LIN {X 0,Y 159.655,Z 246.424,A -85,B 0,C 180,E1 -24975.112,E2 -24975.112} C_VEL
LIN {X 0,Y 158.924,Z 240.028,A -85,B 0,C 180,E1 -24975.712,E2 -24975.712} C_VEL
LIN {X 0,Y 153.683,Z 225.651,A -85,B 0,C 180,E1 -24978.228,E2 -24978.228} C_VEL
LIN {X 0,Y 148.103,Z 213.13,A -85,B 0,C 180,E1 -24981.025,E2 -24981.025} C_VEL
LIN {X 0,Y 143.177,Z 203.296,A -85,B 0,C 180,E1 -24983.678,E2 -24983.678} C_VEL
LIN {X 0,Y 138.265,Z 196.056,A -85,B 0,C 180,E1 -24986.422,E2 -24986.422} C_VEL
LIN {X 0,Y 135.412,Z 191.871,A -85,B 0,C 180,E1 -24988.182,E2 -24988.182} C_VEL
LIN {X 0,Y 133.218,Z 189.003,A -85,B 0,C 180,E1 -24989.591,E2 -24989.591} C_VEL
LIN {X 0,Y 132.456,Z 187.662,A -85,B 0,C 180,E1 -24990.128,E2 -24990.128} C_VEL
LIN {X 0,Y 130.232,Z 185.523,A -85,B 0,C 180,E1 -24991.598,E2 -24991.598} C_VEL
LIN {X 0,Y 129.202,Z 183.065,A -85,B 0,C 180,E1 -24992.458,E2 -24992.458} C_VEL
LIN {X 0,Y 129.076,Z 182.407,A -85,B 0,C 180,E1 -24992.648,E2 -24992.648} C_VEL
LIN {X 0,Y 129.075,Z 182.406,A -85,B 0,C 180,E1 -24997.767,E2 -24997.767} C_VEL
LIN {X 0,Y 129.152,Z 182.398,A -85,B 0,C 180,E1 -25004.209,E2 -25004.209} C_VEL
LIN {X 0,Y 129.347,Z 182.367,A -85,B 0,C 180,E1 -25007.969,E2 -25007.969} C_VEL
LIN {X 0,Y 129.465,Z 182.323,A -85,B 0,C 180,E1 -25010.625,E2 -25010.625} C_VEL
LIN {X 0,Y 130.07,Z 182.267,A -85,B 0,C 180,E1 -25019.997,E2 -25019.997} C_VEL
LIN {X 0,Y 129.471,Z 182.358,A -85,B 0,C 180,E1 -25029.37,E2 -25029.37} C_VEL
LIN {X 0,Y 129.298,Z 182.357,A -85,B 0,C 180,E1 -25032.555,E2 -25032.555} C_VEL
LIN {X 0,Y 129.079,Z 182.388,A -85,B 0,C 180,E1 -25039.065,E2 -25039.065} C_VEL
LIN {X 0,Y 129.034,Z 182.411,A -85,B 0,C 180,E1 -25042.409,E2 -25042.409} C_VEL
LIN {X 0,Y 128.998,Z 182.384,A -85,B 0,C 180,E1 -25049.359,E2 -25049.359} C_VEL
LIN {X 0,Y 128.953,Z 182.408,A -85,B 0,C 180,E1 -25055.163,E2 -25055.163} C_VEL
LIN {X 0,Y 128.92,Z 182.411,A -85,B 0,C 180,E1 -25060.853,E2 -25060.853} C_VEL
LIN {X 0,Y 128.912,Z 182.413,A -85,B 0,C 180,E1 -25065.128,E2 -25065.128} C_VEL
LIN {X 0,Y 128.936,Z 182.51,A -85,B 0,C 180,E1 -25069.928,E2 -25069.928} C_VEL
LIN {X 0,Y 129.826,Z 185.012,A -85,B 0,C 180,E1 -25070.721,E2 -25070.721} C_VEL
LIN {X 0,Y 131.714,Z 187.195,A -85,B 0,C 180,E1 -25072.029,E2 -25072.029} C_VEL
LIN {X 0,Y 132.657,Z 187.914,A -85,B 0,C 180,E1 -25072.621,E2 -25072.621} C_VEL
LIN {X 0,Y 134.637,Z 191.193,A -85,B 0,C 180,E1 -25073.968,E2 -25073.968} C_VEL
LIN {X 0,Y 136.407,Z 193.227,A -85,B 0,C 180,E1 -25075.039,E2 -25075.039} C_VEL
LIN {X 0,Y 140.232,Z 198.848,A -85,B 0,C 180,E1 -25077.317,E2 -25077.317} C_VEL
LIN {X 0,Y 146.175,Z 207.862,A -85,B 0,C 180,E1 -25080.474,E2 -25080.474} C_VEL
LIN {X 0,Y 153.307,Z 220.401,A -85,B 0,C 180,E1 -25083.913,E2 -25083.913} C_VEL
LIN {X 0,Y 160.12,Z 234.099,A -85,B 0,C 180,E1 -25086.884,E2 -25086.884} C_VEL
LIN {X 0,Y 160.428,Z 235.141,A -85,B 0,C 180,E1 -25087.037,E2 -25087.037} C_VEL
LIN {X 0,Y 157.229,Z 278.51,A -85,B 0,C 180,E1 -25088.799,E2 -25088.799} C_VEL
LIN {X 0,Y 155.482,Z 291.667,A -85,B 0,C 180,E1 -25089.752,E2 -25089.752} C_VEL
LIN {X 0,Y 153.102,Z 304.956,A -85,B 0,C 180,E1 -25091.256,E2 -25091.256} C_VEL
LIN {X 0,Y 150.375,Z 316.232,A -85,B 0,C 180,E1 -25093.015,E2 -25093.015} C_VEL
LIN {X 0,Y 146.832,Z 328.024,A -85,B 0,C 180,E1 -25095.446,E2 -25095.446} C_VEL
LIN {X 0,Y 143.106,Z 338.68,A -85,B 0,C 180,E1 -25098.325,E2 -25098.325} C_VEL
LIN {X 0,Y 139.815,Z 347.262,A -85,B 0,C 180,E1 -25101.326,E2 -25101.326} C_VEL
LIN {X 0,Y 135.843,Z 356.621,A -85,B 0,C 180,E1 -25105.548,E2 -25105.548} C_VEL
LIN {X 0,Y 132.556,Z 364.142,A -85,B 0,C 180,E1 -25109.999,E2 -25109.999} C_VEL
LIN {X 0,Y 129.965,Z 370.1,A -85,B 0,C 180,E1 -25114.652,E2 -25114.652} C_VEL
LIN {X 0,Y 128.077,Z 374.766,A -85,B 0,C 180,E1 -25119.475,E2 -25119.475} C_VEL
LIN {X 0,Y 126.764,Z 378.294,A -85,B 0,C 180,E1 -25124.447,E2 -25124.447} C_VEL
LIN {X 0,Y 126.14,Z 380.744,A -85,B 0,C 180,E1 -25129.529,E2 -25129.529} C_VEL
LIN {X 0,Y 126.068,Z 381.808,A -85,B 0,C 180,E1 -25132.969,E2 -25132.969} C_VEL
LIN {X 0,Y 126.473,Z 382.484,A -85,B 0,C 180,E1 -25137.245,E2 -25137.245} C_VEL
LIN {X 0,Y 127.946,Z 382.237,A -85,B 0,C 180,E1 -25143.318,E2 -25143.318} C_VEL
LIN {X 0,Y 129.249,Z 381.455,A -85,B 0,C 180,E1 -25146.736,E2 -25146.736} C_VEL
LIN {X 0,Y 132.014,Z 379.288,A -85,B 0,C 180,E1 -25151.818,E2 -25151.818} C_VEL
LIN {X 0,Y 135.476,Z 376.037,A -85,B 0,C 180,E1 -25156.574,E2 -25156.574} C_VEL
LIN {X 0,Y 139.87,Z 371.452,A -85,B 0,C 180,E1 -25161.152,E2 -25161.152} C_VEL
LIN {X 0,Y 145.081,Z 365.44,A -85,B 0,C 180,E1 -25165.437,E2 -25165.437} C_VEL
LIN {X 0,Y 150.521,Z 358.421,A -85,B 0,C 180,E1 -25169.099,E2 -25169.099} C_VEL
LIN {X 0,Y 156.498,Z 349.628,A -85,B 0,C 180,E1 -25172.49,E2 -25172.49} C_VEL
LIN {X 0,Y 162.372,Z 339.672,A -85,B 0,C 180,E1 -25175.36,E2 -25175.36} C_VEL
LIN {X 0,Y 167.706,Z 328.858,A -85,B 0,C 180,E1 -25177.683,E2 -25177.683} C_VEL
LIN {X 0,Y 172.502,Z 317.181,A -85,B 0,C 180,E1 -25179.562,E2 -25179.562} C_VEL
LIN {X 0,Y 176.144,Z 305.968,A -85,B 0,C 180,E1 -25180.928,E2 -25180.928} C_VEL
LIN {X 0,Y 179.296,Z 292.893,A -85,B 0,C 180,E1 -25182.088,E2 -25182.088} C_VEL
LIN {X 0,Y 181.507,Z 279.685,A -85,B 0,C 180,E1 -25182.847,E2 -25182.847} C_VEL
LIN {X 0,Y 184.072,Z 251.57,A -85,B 0,C 180,E1 -25183.842,E2 -25183.842} C_VEL
LIN {X 0,Y 180.018,Z 243.39,A -85,B 0,C 180,E1 -25186.893,E2 -25186.893} C_VEL
LIN {X 0,Y 175.983,Z 236.11,A -85,B 0,C 180,E1 -25190.417,E2 -25190.417} C_VEL
LIN {X 0,Y 173.194,Z 231.642,A -85,B 0,C 180,E1 -25193.284,E2 -25193.284} C_VEL
LIN {X 0,Y 171.126,Z 228.147,A -85,B 0,C 180,E1 -25195.88,E2 -25195.88} C_VEL
LIN {X 0,Y 168.802,Z 224.365,A -85,B 0,C 180,E1 -25199.501,E2 -25199.501} C_VEL
LIN {X 0,Y 167.756,Z 223.061,A -85,B 0,C 180,E1 -25201.581,E2 -25201.581} C_VEL
LIN {X 0,Y 165.94,Z 219.217,A -85,B 0,C 180,E1 -25208.92,E2 -25208.92} C_VEL
LIN {X 0,Y 165.851,Z 219.507,A -85,B 0,C 180,E1 -25212.018,E2 -25212.018} C_VEL
LIN {X 0,Y 167.881,Z 223.932,A -85,B 0,C 180,E1 -25220.383,E2 -25220.383} C_VEL
LIN {X 0,Y 168.683,Z 224.803,A -85,B 0,C 180,E1 -25221.922,E2 -25221.922} C_VEL
LIN {X 0,Y 170.864,Z 228.31,A -85,B 0,C 180,E1 -25225.363,E2 -25225.363} C_VEL
LIN {X 0,Y 171.907,Z 230.371,A -85,B 0,C 180,E1 -25226.809,E2 -25226.809} C_VEL
LIN {X 0,Y 174.118,Z 234.701,A -85,B 0,C 180,E1 -25229.416,E2 -25229.416} C_VEL
LIN {X 0,Y 176.962,Z 240.729,A -85,B 0,C 180,E1 -25232.329,E2 -25232.329} C_VEL
LIN {X 0,Y 180.022,Z 248.005,A -85,B 0,C 180,E1 -25235.04,E2 -25235.04} C_VEL
LIN {X 0,Y 183.032,Z 256.153,A -85,B 0,C 180,E1 -25237.487,E2 -25237.487} C_VEL
LIN {X 0,Y 183.665,Z 258.053,A -85,B 0,C 180,E1 -25237.971,E2 -25237.971} C_VEL
LIN {X 0,Y 180.889,Z 287.544,A -85,B 0,C 180,E1 -25239.009,E2 -25239.009} C_VEL
LIN {X 0,Y 178.421,Z 301.333,A -85,B 0,C 180,E1 -25239.796,E2 -25239.796} C_VEL
LIN {X 0,Y 175.156,Z 313.446,A -85,B 0,C 180,E1 -25240.77,E2 -25240.77} C_VEL
LIN {X 0,Y 170.748,Z 325.878,A -85,B 0,C 180,E1 -25242.194,E2 -25242.194} C_VEL
LIN {X 0,Y 165.903,Z 337.01,A -85,B 0,C 180,E1 -25243.933,E2 -25243.933} C_VEL
LIN {X 0,Y 160.841,Z 347.084,A -85,B 0,C 180,E1 -25246.08,E2 -25246.08} C_VEL
LIN {X 0,Y 154.847,Z 357.022,A -85,B 0,C 180,E1 -25248.845,E2 -25248.845} C_VEL
LIN {X 0,Y 148.836,Z 365.808,A -85,B 0,C 180,E1 -25252.132,E2 -25252.132} C_VEL
LIN {X 0,Y 143.478,Z 372.904,A -85,B 0,C 180,E1 -25255.716,E2 -25255.716} C_VEL
LIN {X 0,Y 138.921,Z 378.614,A -85,B 0,C 180,E1 -25259.609,E2 -25259.609} C_VEL
LIN {X 0,Y 134.806,Z 383.156,A -85,B 0,C 180,E1 -25263.696,E2 -25263.696} C_VEL
LIN {X 0,Y 131.486,Z 386.642,A -85,B 0,C 180,E1 -25268.029,E2 -25268.029} C_VEL
LIN {X 0,Y 129.685,Z 388.403,A -85,B 0,C 180,E1 -25271.025,E2 -25271.025} C_VEL
LIN {X 0,Y 127.395,Z 390.753,A -85,B 0,C 180,E1 -25277.252,E2 -25277.252} C_VEL
LIN {X 0,Y 126.764,Z 391.356,A -85,B 0,C 180,E1 -25280.426,E2 -25280.426} C_VEL
LIN {X 0,Y 126.378,Z 391.329,A -85,B 0,C 180,E1 -25286.813,E2 -25286.813} C_VEL
LIN {X 0,Y 126.519,Z 390.56,A -85,B 0,C 180,E1 -25290.716,E2 -25290.716} C_VEL
LIN {X 0,Y 126.472,Z 388.249,A -85,B 0,C 180,E1 -25296.382,E2 -25296.382} C_VEL
LIN {X 0,Y 127.056,Z 385.219,A -85,B 0,C 180,E1 -25301.164,E2 -25301.164} C_VEL
LIN {X 0,Y 128.223,Z 381.214,A -85,B 0,C 180,E1 -25305.777,E2 -25305.777} C_VEL
LIN {X 0,Y 128.498,Z 378.783,A -85,B 0,C 180,E1 -25308.176,E2 -25308.176} C_VEL
LIN {X 0,Y 127.692,Z 374.194,A -85,B 0,C 180,E1 -25312.083,E2 -25312.083} C_VEL
LIN {X 0,Y 127.184,Z 368.915,A -85,B 0,C 180,E1 -25315.87,E2 -25315.87} C_VEL
LIN {X 0,Y 127.915,Z 365.396,A -85,B 0,C 180,E1 -25317.996,E2 -25317.996} C_VEL
LIN {X 0,Y 131.866,Z 356.514,A -85,B 0,C 180,E1 -25322.207,E2 -25322.207} C_VEL
LIN {X 0,Y 135.805,Z 347.059,A -85,B 0,C 180,E1 -25325.606,E2 -25325.606} C_VEL
LIN {X 0,Y 139.802,Z 336.564,A -85,B 0,C 180,E1 -25328.471,E2 -25328.471} C_VEL
LIN {X 0,Y 143.139,Z 326.497,A -85,B 0,C 180,E1 -25330.585,E2 -25330.585} C_VEL
LIN {X 0,Y 146.471,Z 314.751,A -85,B 0,C 180,E1 -25332.436,E2 -25332.436} C_VEL
LIN {X 0,Y 149.169,Z 301.868,A -85,B 0,C 180,E1 -25333.906,E2 -25333.906} C_VEL
LIN {X 0,Y 151.169,Z 288.247,A -85,B 0,C 180,E1 -25334.921,E2 -25334.921} C_VEL
LIN {X 0,Y 154.109,Z 247.24,A -85,B 0,C 180,E1 -25336.713,E2 -25336.713} C_VEL
LIN {X 0,Y 153.578,Z 242.635,A -85,B 0,C 180,E1 -25337.17,E2 -25337.17} C_VEL
LIN {X 0,Y 148.756,Z 229.08,A -85,B 0,C 180,E1 -25339.679,E2 -25339.679} C_VEL
LIN {X 0,Y 142.765,Z 215.286,A -85,B 0,C 180,E1 -25342.947,E2 -25342.947} C_VEL
LIN {X 0,Y 138.609,Z 207.245,A -85,B 0,C 180,E1 -25345.356,E2 -25345.356} C_VEL
LIN {X 0,Y 134.487,Z 201.113,A -85,B 0,C 180,E1 -25347.856,E2 -25347.856} C_VEL
LIN {X 0,Y 131.979,Z 197.416,A -85,B 0,C 180,E1 -25349.497,E2 -25349.497} C_VEL
LIN {X 0,Y 129.155,Z 193.437,A -85,B 0,C 180,E1 -25351.469,E2 -25351.469} C_VEL
LIN {X 0,Y 126.841,Z 190.647,A -85,B 0,C 180,E1 -25353.176,E2 -25353.176} C_VEL
LIN {X 0,Y 125.964,Z 188.807,A -85,B 0,C 180,E1 -25353.933,E2 -25353.933} C_VEL
LIN {X 0,Y 123.487,Z 186.896,A -85,B 0,C 180,E1 -25355.851,E2 -25355.851} C_VEL
LIN {X 0,Y 122.221,Z 184.395,A -85,B 0,C 180,E1 -25357.08,E2 -25357.08} C_VEL
LIN {X 0,Y 122.024,Z 183.284,A -85,B 0,C 180,E1 -25357.449,E2 -25357.449} C_VEL
LIN {X 0,Y 122.065,Z 183.28,A -85,B 0,C 180,E1 -25363.266,E2 -25363.266} C_VEL
LIN {X 0,Y 122.29,Z 183.248,A -85,B 0,C 180,E1 -25367.689,E2 -25367.689} C_VEL
LIN {X 0,Y 122.394,Z 183.207,A -85,B 0,C 180,E1 -25370.078,E2 -25370.078} C_VEL
LIN {X 0,Y 122.565,Z 183.215,A -85,B 0,C 180,E1 -25376.71,E2 -25376.71} C_VEL
LIN {X 0,Y 123.023,Z 183.142,A -85,B 0,C 180,E1 -25379.997,E2 -25379.997} C_VEL
LIN {X 0,Y 122.392,Z 183.215,A -85,B 0,C 180,E1 -25386.899,E2 -25386.899} C_VEL
LIN {X 0,Y 122.288,Z 183.231,A -85,B 0,C 180,E1 -25392.305,E2 -25392.305} C_VEL
LIN {X 0,Y 122.057,Z 183.236,A -85,B 0,C 180,E1 -25396.729,E2 -25396.729} C_VEL
LIN {X 0,Y 121.978,Z 183.287,A -85,B 0,C 180,E1 -25402.797,E2 -25402.797} C_VEL
LIN {X 0,Y 121.914,Z 183.273,A -85,B 0,C 180,E1 -25410.149,E2 -25410.149} C_VEL
LIN {X 0,Y 121.878,Z 183.276,A -85,B 0,C 180,E1 -25416.165,E2 -25416.165} C_VEL
LIN {X 0,Y 121.861,Z 183.296,A -85,B 0,C 180,E1 -25421.431,E2 -25421.431} C_VEL
LIN {X 0,Y 121.884,Z 183.332,A -85,B 0,C 180,E1 -25425.152,E2 -25425.152} C_VEL
LIN {X 0,Y 122.547,Z 185.608,A -85,B 0,C 180,E1 -25425.92,E2 -25425.92} C_VEL
LIN {X 0,Y 124.203,Z 187.76,A -85,B 0,C 180,E1 -25427.354,E2 -25427.354} C_VEL
LIN {X 0,Y 125.952,Z 189.095,A -85,B 0,C 180,E1 -25428.69,E2 -25428.69} C_VEL
LIN {X 0,Y 127.916,Z 192.295,A -85,B 0,C 180,E1 -25430.277,E2 -25430.277} C_VEL
LIN {X 0,Y 129.731,Z 194.29,A -85,B 0,C 180,E1 -25431.564,E2 -25431.564} C_VEL
LIN {X 0,Y 132.223,Z 197.774,A -85,B 0,C 180,E1 -25433.284,E2 -25433.284} C_VEL
LIN {X 0,Y 136.409,Z 203.859,A -85,B 0,C 180,E1 -25435.94,E2 -25435.94} C_VEL
LIN {X 0,Y 142.242,Z 212.947,A -85,B 0,C 180,E1 -25439.276,E2 -25439.276} C_VEL
LIN {X 0,Y 148.873,Z 224.925,A -85,B 0,C 180,E1 -25442.683,E2 -25442.683} C_VEL
LIN {X 0,Y 154.802,Z 237.212,A -85,B 0,C 180,E1 -25445.478,E2 -25445.478} C_VEL
LIN {X 0,Y 151.462,Z 279.808,A -85,B 0,C 180,E1 -25447.259,E2 -25447.259} C_VEL
LIN {X 0,Y 149.487,Z 293.866,A -85,B 0,C 180,E1 -25448.36,E2 -25448.36} C_VEL
LIN {X 0,Y 146.973,Z 306.542,A -85,B 0,C 180,E1 -25449.897,E2 -25449.897} C_VEL
LIN {X 0,Y 143.903,Z 318.341,A -85,B 0,C 180,E1 -25451.859,E2 -25451.859} C_VEL
LIN {X 0,Y 140.242,Z 329.793,A -85,B 0,C 180,E1 -25454.373,E2 -25454.373} C_VEL
LIN {X 0,Y 136.133,Z 340.779,A -85,B 0,C 180,E1 -25457.6,E2 -25457.6} C_VEL
LIN {X 0,Y 131.879,Z 351.007,A -85,B 0,C 180,E1 -25461.572,E2 -25461.572} C_VEL
LIN {X 0,Y 127.91,Z 359.66,A -85,B 0,C 180,E1 -25466.061,E2 -25466.061} C_VEL
LIN {X 0,Y 124.714,Z 366.598,A -85,B 0,C 180,E1 -25470.807,E2 -25470.807} C_VEL
LIN {X 0,Y 122.596,Z 371.268,A -85,B 0,C 180,E1 -25474.932,E2 -25474.932} C_VEL
LIN {X 0,Y 120.726,Z 375.736,A -85,B 0,C 180,E1 -25480.057,E2 -25480.057} C_VEL
LIN {X 0,Y 119.836,Z 378.103,A -85,B 0,C 180,E1 -25483.567,E2 -25483.567} C_VEL
LIN {X 0,Y 119.067,Z 380.811,A -85,B 0,C 180,E1 -25489.204,E2 -25489.204} C_VEL
LIN {X 0,Y 119.042,Z 382.299,A -85,B 0,C 180,E1 -25494.41,E2 -25494.41} C_VEL
LIN {X 0,Y 119.507,Z 382.759,A -85,B 0,C 180,E1 -25498.107,E2 -25498.107} C_VEL
LIN {X 0,Y 120.282,Z 382.786,A -85,B 0,C 180,E1 -25501.726,E2 -25501.726} C_VEL
LIN {X 0,Y 121.785,Z 382.173,A -85,B 0,C 180,E1 -25506.112,E2 -25506.112} C_VEL
LIN {X 0,Y 125.032,Z 380.001,A -85,B 0,C 180,E1 -25512.416,E2 -25512.416} C_VEL
LIN {X 0,Y 128.74,Z 376.916,A -85,B 0,C 180,E1 -25517.474,E2 -25517.474} C_VEL
LIN {X 0,Y 133.332,Z 372.545,A -85,B 0,C 180,E1 -25522.246,E2 -25522.246} C_VEL
LIN {X 0,Y 138.964,Z 366.536,A -85,B 0,C 180,E1 -25526.824,E2 -25526.824} C_VEL
LIN {X 0,Y 144.969,Z 359.35,A -85,B 0,C 180,E1 -25530.765,E2 -25530.765} C_VEL
LIN {X 0,Y 150.642,Z 351.6,A -85,B 0,C 180,E1 -25533.906,E2 -25533.906} C_VEL
LIN {X 0,Y 156.459,Z 342.417,A -85,B 0,C 180,E1 -25536.721,E2 -25536.721} C_VEL
LIN {X 0,Y 161.839,Z 332.55,A -85,B 0,C 180,E1 -25539.012,E2 -25539.012} C_VEL
LIN {X 0,Y 166.518,Z 322.467,A -85,B 0,C 180,E1 -25540.795,E2 -25540.795} C_VEL
LIN {X 0,Y 170.526,Z 311.872,A -85,B 0,C 180,E1 -25542.261,E2 -25542.261} C_VEL
LIN {X 0,Y 174.114,Z 299.664,A -85,B 0,C 180,E1 -25543.518,E2 -25543.518} C_VEL
LIN {X 0,Y 176.92,Z 286.36,A -85,B 0,C 180,E1 -25544.477,E2 -25544.477} C_VEL
LIN {X 0,Y 178.669,Z 273.562,A -85,B 0,C 180,E1 -25545.007,E2 -25545.007} C_VEL
LIN {X 0,Y 180.308,Z 255.055,A -85,B 0,C 180,E1 -25545.666,E2 -25545.666} C_VEL
LIN {X 0,Y 177.07,Z 248.273,A -85,B 0,C 180,E1 -25548.343,E2 -25548.343} C_VEL
LIN {X 0,Y 173.689,Z 241.928,A -85,B 0,C 180,E1 -25551.594,E2 -25551.594} C_VEL
LIN {X 0,Y 171.438,Z 238.08,A -85,B 0,C 180,E1 -25554.1,E2 -25554.1} C_VEL
LIN {X 0,Y 169.428,Z 234.559,A -85,B 0,C 180,E1 -25556.829,E2 -25556.829} C_VEL
LIN {X 0,Y 167.24,Z 230.626,A -85,B 0,C 180,E1 -25560.679,E2 -25560.679} C_VEL
LIN {X 0,Y 164.992,Z 226.368,A -85,B 0,C 180,E1 -25568.972,E2 -25568.972} C_VEL
LIN {X 0,Y 164.907,Z 226.471,A -85,B 0,C 180,E1 -25571.649,E2 -25571.649} C_VEL
LIN {X 0,Y 166.862,Z 230.946,A -85,B 0,C 180,E1 -25580.239,E2 -25580.239} C_VEL
LIN {X 0,Y 167.452,Z 231.73,A -85,B 0,C 180,E1 -25581.451,E2 -25581.451} C_VEL
LIN {X 0,Y 169.788,Z 235.723,A -85,B 0,C 180,E1 -25585.295,E2 -25585.295} C_VEL
LIN {X 0,Y 172.252,Z 241.088,A -85,B 0,C 180,E1 -25588.566,E2 -25588.566} C_VEL
LIN {X 0,Y 174.858,Z 246.961,A -85,B 0,C 180,E1 -25591.424,E2 -25591.424} C_VEL
LIN {X 0,Y 177.667,Z 254.325,A -85,B 0,C 180,E1 -25594.143,E2 -25594.143} C_VEL
LIN {X 0,Y 179.895,Z 260.761,A -85,B 0,C 180,E1 -25596.103,E2 -25596.103} C_VEL
LIN {X 0,Y 177.174,Z 288.011,A -85,B 0,C 180,E1 -25597.081,E2 -25597.081} C_VEL
LIN {X 0,Y 174.578,Z 301.687,A -85,B 0,C 180,E1 -25597.863,E2 -25597.863} C_VEL
LIN {X 0,Y 171.321,Z 313.255,A -85,B 0,C 180,E1 -25598.792,E2 -25598.792} C_VEL
LIN {X 0,Y 166.761,Z 325.643,A -85,B 0,C 180,E1 -25600.194,E2 -25600.194} C_VEL
LIN {X 0,Y 161.697,Z 336.776,A -85,B 0,C 180,E1 -25601.9,E2 -25601.9} C_VEL
LIN {X 0,Y 156.44,Z 346.839,A -85,B 0,C 180,E1 -25604.045,E2 -25604.045} C_VEL
LIN {X 0,Y 150.721,Z 355.965,A -85,B 0,C 180,E1 -25606.546,E2 -25606.546} C_VEL
LIN {X 0,Y 144.313,Z 364.887,A -85,B 0,C 180,E1 -25609.814,E2 -25609.814} C_VEL
LIN {X 0,Y 138.559,Z 372.104,A -85,B 0,C 180,E1 -25613.418,E2 -25613.418} C_VEL
LIN {X 0,Y 132.826,Z 378.747,A -85,B 0,C 180,E1 -25618.055,E2 -25618.055} C_VEL
LIN {X 0,Y 128.467,Z 383.188,A -85,B 0,C 180,E1 -25622.29,E2 -25622.29} C_VEL
LIN {X 0,Y 124.918,Z 386.594,A -85,B 0,C 180,E1 -25626.808,E2 -25626.808} C_VEL
LIN {X 0,Y 122.968,Z 388.312,A -85,B 0,C 180,E1 -25629.946,E2 -25629.946} C_VEL
LIN {X 0,Y 120.461,Z 390.586,A -85,B 0,C 180,E1 -25636.505,E2 -25636.505} C_VEL
LIN {X 0,Y 119.734,Z 391.124,A -85,B 0,C 180,E1 -25639.858,E2 -25639.858} C_VEL
LIN {X 0,Y 119.284,Z 391.012,A -85,B 0,C 180,E1 -25646.623,E2 -25646.623} C_VEL
LIN {X 0,Y 119.481,Z 390.384,A -85,B 0,C 180,E1 -25650.001,E2 -25650.001} C_VEL
LIN {X 0,Y 119.296,Z 389.315,A -85,B 0,C 180,E1 -25653.378,E2 -25653.378} C_VEL
LIN {X 0,Y 119.419,Z 387.786,A -85,B 0,C 180,E1 -25656.76,E2 -25656.76} C_VEL
LIN {X 0,Y 120.068,Z 384.676,A -85,B 0,C 180,E1 -25661.823,E2 -25661.823} C_VEL
LIN {X 0,Y 121.398,Z 380.467,A -85,B 0,C 180,E1 -25666.827,E2 -25666.827} C_VEL
LIN {X 0,Y 124.169,Z 374.049,A -85,B 0,C 180,E1 -25672.462,E2 -25672.462} C_VEL
LIN {X 0,Y 127.265,Z 367.194,A -85,B 0,C 180,E1 -25676.985,E2 -25676.985} C_VEL
LIN {X 0,Y 127.915,Z 365.396,A -85,B 0,C 180,E1 -25677.996,E2 -25677.996} C_VEL
LIN {X 0,Y 128.739,Z 361.719,A -85,B 0,C 180,E1 -25680.028,E2 -25680.028} C_VEL
LIN {X 0,Y 128.916,Z 355.288,A -85,B 0,C 180,E1 -25683.383,E2 -25683.383} C_VEL
LIN {X 0,Y 129.481,Z 348.333,A -85,B 0,C 180,E1 -25686.495,E2 -25686.495} C_VEL
LIN {X 0,Y 130.848,Z 343.784,A -85,B 0,C 180,E1 -25688.07,E2 -25688.07} C_VEL
LIN {X 0,Y 134.817,Z 333.764,A -85,B 0,C 180,E1 -25690.665,E2 -25690.665} C_VEL
LIN {X 0,Y 138.25,Z 323.003,A -85,B 0,C 180,E1 -25692.839,E2 -25692.839} C_VEL
LIN {X 0,Y 141.829,Z 310.18,A -85,B 0,C 180,E1 -25694.672,E2 -25694.672} C_VEL
LIN {X 0,Y 144.409,Z 297.139,A -85,B 0,C 180,E1 -25696.003,E2 -25696.003} C_VEL
LIN {X 0,Y 146.052,Z 283.861,A -85,B 0,C 180,E1 -25696.868,E2 -25696.868} C_VEL
LIN {X 0,Y 148.645,Z 248.086,A -85,B 0,C 180,E1 -25698.426,E2 -25698.426} C_VEL
LIN {X 0,Y 148.205,Z 244.825,A -85,B 0,C 180,E1 -25698.798,E2 -25698.798} C_VEL
LIN {X 0,Y 143.705,Z 231.939,A -85,B 0,C 180,E1 -25701.353,E2 -25701.353} C_VEL
LIN {X 0,Y 137.967,Z 218.512,A -85,B 0,C 180,E1 -25704.741,E2 -25704.741} C_VEL
LIN {X 0,Y 134.475,Z 211.629,A -85,B 0,C 180,E1 -25706.955,E2 -25706.955} C_VEL
LIN {X 0,Y 128.632,Z 202.898,A -85,B 0,C 180,E1 -25710.862,E2 -25710.862} C_VEL
LIN {X 0,Y 125.808,Z 198.989,A -85,B 0,C 180,E1 -25712.98,E2 -25712.98} C_VEL
LIN {X 0,Y 123.328,Z 195.401,A -85,B 0,C 180,E1 -25715.026,E2 -25715.026} C_VEL
LIN {X 0,Y 120.234,Z 192,A -85,B 0,C 180,E1 -25717.713,E2 -25717.713} C_VEL
LIN {X 0,Y 119.181,Z 189.797,A -85,B 0,C 180,E1 -25718.836,E2 -25718.836} C_VEL
LIN {X 0,Y 116.544,Z 187.838,A -85,B 0,C 180,E1 -25721.426,E2 -25721.426} C_VEL
LIN {X 0,Y 115.305,Z 185.539,A -85,B 0,C 180,E1 -25722.94,E2 -25722.94} C_VEL
LIN {X 0,Y 115.024,Z 184.158,A -85,B 0,C 180,E1 -25723.582,E2 -25723.582} C_VEL
LIN {X 0,Y 115.308,Z 184.093,A -85,B 0,C 180,E1 -25729.461,E2 -25729.461} C_VEL
LIN {X 0,Y 115.491,Z 184.095,A -85,B 0,C 180,E1 -25736.508,E2 -25736.508} C_VEL
LIN {X 0,Y 115.975,Z 184.018,A -85,B 0,C 180,E1 -25739.997,E2 -25739.997} C_VEL
LIN {X 0,Y 115.352,Z 184.095,A -85,B 0,C 180,E1 -25746.996,E2 -25746.996} C_VEL
LIN {X 0,Y 115.204,Z 184.107,A -85,B 0,C 180,E1 -25752.554,E2 -25752.554} C_VEL
LIN {X 0,Y 114.962,Z 184.126,A -85,B 0,C 180,E1 -25757.795,E2 -25757.795} C_VEL
LIN {X 0,Y 114.892,Z 184.163,A -85,B 0,C 180,E1 -25763.426,E2 -25763.426} C_VEL
LIN {X 0,Y 114.845,Z 184.164,A -85,B 0,C 180,E1 -25771.046,E2 -25771.046} C_VEL
LIN {X 0,Y 114.771,Z 184.152,A -85,B 0,C 180,E1 -25777.756,E2 -25777.756} C_VEL
LIN {X 0,Y 114.798,Z 184.167,A -85,B 0,C 180,E1 -25778.933,E2 -25778.933} C_VEL
LIN {X 0,Y 115.586,Z 186.624,A -85,B 0,C 180,E1 -25780.097,E2 -25780.097} C_VEL
LIN {X 0,Y 117.601,Z 188.973,A -85,B 0,C 180,E1 -25782.31,E2 -25782.31} C_VEL
LIN {X 0,Y 119.13,Z 189.955,A -85,B 0,C 180,E1 -25783.758,E2 -25783.758} C_VEL
LIN {X 0,Y 120.811,Z 193.04,A -85,B 0,C 180,E1 -25785.478,E2 -25785.478} C_VEL
LIN {X 0,Y 123.234,Z 195.428,A -85,B 0,C 180,E1 -25787.52,E2 -25787.52} C_VEL
LIN {X 0,Y 125.859,Z 199.11,A -85,B 0,C 180,E1 -25789.673,E2 -25789.673} C_VEL
LIN {X 0,Y 130.257,Z 205.284,A -85,B 0,C 180,E1 -25792.9,E2 -25792.9} C_VEL
LIN {X 0,Y 134.7,Z 211.987,A -85,B 0,C 180,E1 -25795.792,E2 -25795.792} C_VEL
LIN {X 0,Y 140.152,Z 221.297,A -85,B 0,C 180,E1 -25799.038,E2 -25799.038} C_VEL
LIN {X 0,Y 145.492,Z 231.35,A -85,B 0,C 180,E1 -25801.891,E2 -25801.891} C_VEL
LIN {X 0,Y 149.229,Z 239.356,A -85,B 0,C 180,E1 -25803.79,E2 -25803.79} C_VEL
